LIN {X 0,Y 473.859,Z 535.178,A -85,B 0,C 180,E1 -7292.55,E2 -7292.55} C_VEL
LIN {X 0,Y 473.786,Z 533.185,A -85,B 0,C 180,E1 -7294.253,E2 -7294.253} C_VEL
LIN {X 0,Y 473.862,Z 529.069,A -85,B 0,C 180,E1 -7296.438,E2 -7296.438} C_VEL
LIN {X 0,Y 473.899,Z 524.706,A -85,B 0,C 180,E1 -7298.099,E2 -7298.099} C_VEL
LIN {X 0,Y 473.982,Z 519.093,A -85,B 0,C 180,E1 -7299.817,E2 -7299.817} C_VEL
LIN {X 0,Y 474.226,Z 512.098,A -85,B 0,C 180,E1 -7301.54,E2 -7301.54} C_VEL
LIN {X 0,Y 474.535,Z 503.681,A -85,B 0,C 180,E1 -7303.271,E2 -7303.271} C_VEL
LIN {X 0,Y 475.075,Z 493.63,A -85,B 0,C 180,E1 -7305.003,E2 -7305.003} C_VEL
LIN {X 0,Y 475.646,Z 483.269,A -85,B 0,C 180,E1 -7306.524,E2 -7306.524} C_VEL
LIN {X 0,Y 476.368,Z 471.017,A -85,B 0,C 180,E1 -7308.048,E2 -7308.048} C_VEL
LIN {X 0,Y 477.233,Z 457.973,A -85,B 0,C 180,E1 -7309.422,E2 -7309.422} C_VEL
LIN {X 0,Y 478.152,Z 444.159,A -85,B 0,C 180,E1 -7310.655,E2 -7310.655} C_VEL
LIN {X 0,Y 479.041,Z 429.731,A -85,B 0,C 180,E1 -7311.742,E2 -7311.742} C_VEL
LIN {X 0,Y 479.978,Z 414.203,A -85,B 0,C 180,E1 -7312.711,E2 -7312.711} C_VEL
LIN {X 0,Y 480.906,Z 398.033,A -85,B 0,C 180,E1 -7313.524,E2 -7313.524} C_VEL
LIN {X 0,Y 481.693,Z 381.393,A -85,B 0,C 180,E1 -7314.169,E2 -7314.169} C_VEL
LIN {X 0,Y 482.3,Z 365.314,A -85,B 0,C 180,E1 -7314.623,E2 -7314.623} C_VEL
LIN {X 0,Y 482.825,Z 343.034,A -85,B 0,C 180,E1 -7315.038,E2 -7315.038} C_VEL
LIN {X 0,Y 485.86,Z 178.498,A -85,B 0,C 180,E1 -7317.853,E2 -7317.853} C_VEL
LIN {X 0,Y 482.039,Z 153.132,A -85,B 0,C 180,E1 -7318.567,E2 -7318.567} C_VEL
LIN {X 0,Y 483.529,Z 126.486,A -85,B 0,C 180,E1 -7321.047,E2 -7321.047} C_VEL
LIN {X 0,Y 482.934,Z 123.424,A -85,B 0,C 180,E1 -7321.381,E2 -7321.381} C_VEL
LIN {X 0,Y 476.541,Z 103.71,A -85,B 0,C 180,E1 -7323.756,E2 -7323.756} C_VEL
LIN {X 0,Y 474.657,Z 97.672,A -85,B 0,C 180,E1 -7324.527,E2 -7324.527} C_VEL
LIN {X 0,Y 474.585,Z 97.681,A -85,B 0,C 180,E1 -7327.383,E2 -7327.383} C_VEL
LIN {X 0,Y 474.623,Z 97.676,A -85,B 0,C 180,E1 -7329.647,E2 -7329.647} C_VEL
LIN {X 0,Y 474.648,Z 97.673,A -85,B 0,C 180,E1 -7332.93,E2 -7332.93} C_VEL
LIN {X 0,Y 474.605,Z 97.678,A -85,B 0,C 180,E1 -7335.895,E2 -7335.895} C_VEL
LIN {X 0,Y 474.623,Z 97.672,A -85,B 0,C 180,E1 -7339.04,E2 -7339.04} C_VEL
LIN {X 0,Y 474.606,Z 97.675,A -85,B 0,C 180,E1 -7341.704,E2 -7341.704} C_VEL
LIN {X 0,Y 474.626,Z 97.674,A -85,B 0,C 180,E1 -7344.726,E2 -7344.726} C_VEL
LIN {X 0,Y 474.632,Z 97.674,A -85,B 0,C 180,E1 -7347.788,E2 -7347.788} C_VEL
LIN {X 0,Y 474.62,Z 97.673,A -85,B 0,C 180,E1 -7350.884,E2 -7350.884} C_VEL
LIN {X 0,Y 474.656,Z 97.67,A -85,B 0,C 180,E1 -7353.628,E2 -7353.628} C_VEL
LIN {X 0,Y 474.631,Z 97.672,A -85,B 0,C 180,E1 -7356.641,E2 -7356.641} C_VEL
LIN {X 0,Y 474.65,Z 97.675,A -85,B 0,C 180,E1 -7360.09,E2 -7360.09} C_VEL
LIN {X 0,Y 474.646,Z 97.669,A -85,B 0,C 180,E1 -7362.774,E2 -7362.774} C_VEL
LIN {X 0,Y 474.644,Z 97.672,A -85,B 0,C 180,E1 -7365.421,E2 -7365.421} C_VEL
LIN {X 0,Y 474.734,Z 97.663,A -85,B 0,C 180,E1 -7368.038,E2 -7368.038} C_VEL
LIN {X 0,Y 474.723,Z 97.663,A -85,B 0,C 180,E1 -7371.487,E2 -7371.487} C_VEL
LIN {X 0,Y 474.774,Z 97.657,A -85,B 0,C 180,E1 -7374.052,E2 -7374.052} C_VEL
LIN {X 0,Y 474.89,Z 97.644,A -85,B 0,C 180,E1 -7377.455,E2 -7377.455} C_VEL
LIN {X 0,Y 474.908,Z 97.64,A -85,B 0,C 180,E1 -7380,E2 -7380} C_VEL
LIN {X 0,Y 474.89,Z 97.638,A -85,B 0,C 180,E1 -7382.545,E2 -7382.545} C_VEL
LIN {X 0,Y 474.774,Z 97.656,A -85,B 0,C 180,E1 -7385.948,E2 -7385.948} C_VEL
LIN {X 0,Y 474.723,Z 97.659,A -85,B 0,C 180,E1 -7388.514,E2 -7388.514} C_VEL
LIN {X 0,Y 474.7,Z 97.664,A -85,B 0,C 180,E1 -7391.963,E2 -7391.963} C_VEL
LIN {X 0,Y 474.696,Z 97.67,A -85,B 0,C 180,E1 -7395.456,E2 -7395.456} C_VEL
LIN {X 0,Y 474.661,Z 97.671,A -85,B 0,C 180,E1 -7399.01,E2 -7399.01} C_VEL
LIN {X 0,Y 474.587,Z 97.679,A -85,B 0,C 180,E1 -7401.729,E2 -7401.729} C_VEL
LIN {X 0,Y 474.655,Z 97.668,A -85,B 0,C 180,E1 -7404.493,E2 -7404.493} C_VEL
LIN {X 0,Y 474.677,Z 97.671,A -85,B 0,C 180,E1 -7407.335,E2 -7407.335} C_VEL
LIN {X 0,Y 474.602,Z 97.674,A -85,B 0,C 180,E1 -7410.23,E2 -7410.23} C_VEL
LIN {X 0,Y 474.639,Z 97.676,A -85,B 0,C 180,E1 -7413.22,E2 -7413.22} C_VEL
LIN {X 0,Y 474.59,Z 97.677,A -85,B 0,C 180,E1 -7416.323,E2 -7416.323} C_VEL
LIN {X 0,Y 474.624,Z 97.672,A -85,B 0,C 180,E1 -7419.648,E2 -7419.648} C_VEL
LIN {X 0,Y 474.637,Z 97.678,A -85,B 0,C 180,E1 -7422.932,E2 -7422.932} C_VEL
LIN {X 0,Y 474.612,Z 97.673,A -85,B 0,C 180,E1 -7425.896,E2 -7425.896} C_VEL
LIN {X 0,Y 474.629,Z 97.676,A -85,B 0,C 180,E1 -7429.041,E2 -7429.041} C_VEL
LIN {X 0,Y 474.607,Z 97.674,A -85,B 0,C 180,E1 -7431.705,E2 -7431.705} C_VEL
LIN {X 0,Y 474.622,Z 97.68,A -85,B 0,C 180,E1 -7434.726,E2 -7434.726} C_VEL
LIN {X 0,Y 474.634,Z 97.671,A -85,B 0,C 180,E1 -7437.788,E2 -7437.788} C_VEL
LIN {X 0,Y 474.622,Z 97.676,A -85,B 0,C 180,E1 -7440.885,E2 -7440.885} C_VEL
LIN {X 0,Y 474.659,Z 97.667,A -85,B 0,C 180,E1 -7443.629,E2 -7443.629} C_VEL
LIN {X 0,Y 474.634,Z 97.676,A -85,B 0,C 180,E1 -7446.642,E2 -7446.642} C_VEL
LIN {X 0,Y 474.654,Z 97.672,A -85,B 0,C 180,E1 -7450.09,E2 -7450.09} C_VEL
LIN {X 0,Y 474.655,Z 97.668,A -85,B 0,C 180,E1 -7451.674,E2 -7451.674} C_VEL
LIN {X 0,Y 473.992,Z 97.759,A -85,B 0,C 180,E1 -7452.383,E2 -7452.383} C_VEL
LIN {X 0,Y 471.141,Z 98.108,A -85,B 0,C 180,E1 -7453.534,E2 -7453.534} C_VEL
LIN {X 0,Y 468.725,Z 98.413,A -85,B 0,C 180,E1 -7454.463,E2 -7454.463} C_VEL
LIN {X 0,Y 467.683,Z 98.537,A -85,B 0,C 180,E1 -7455.18,E2 -7455.18} C_VEL
LIN {X 0,Y 467.596,Z 98.547,A -85,B 0,C 180,E1 -7455.423,E2 -7455.423} C_VEL
LIN {X 0,Y 467.653,Z 98.542,A -85,B 0,C 180,E1 -7458.734,E2 -7458.734} C_VEL
LIN {X 0,Y 467.749,Z 98.536,A -85,B 0,C 180,E1 -7462.229,E2 -7462.229} C_VEL
LIN {X 0,Y 467.724,Z 98.532,A -85,B 0,C 180,E1 -7464.828,E2 -7464.828} C_VEL
LIN {X 0,Y 467.86,Z 98.515,A -85,B 0,C 180,E1 -7467.418,E2 -7467.418} C_VEL
LIN {X 0,Y 467.883,Z 98.519,A -85,B 0,C 180,E1 -7470.001,E2 -7470.001} C_VEL
LIN {X 0,Y 467.86,Z 98.516,A -85,B 0,C 180,E1 -7472.583,E2 -7472.583} C_VEL
LIN {X 0,Y 467.744,Z 98.536,A -85,B 0,C 180,E1 -7476.038,E2 -7476.038} C_VEL
LIN {X 0,Y 467.683,Z 98.537,A -85,B 0,C 180,E1 -7478.643,E2 -7478.643} C_VEL
LIN {X 0,Y 467.658,Z 98.544,A -85,B 0,C 180,E1 -7482.146,E2 -7482.146} C_VEL
LIN {X 0,Y 467.641,Z 98.549,A -85,B 0,C 180,E1 -7485.695,E2 -7485.695} C_VEL
LIN {X 0,Y 467.619,Z 98.544,A -85,B 0,C 180,E1 -7488.765,E2 -7488.765} C_VEL
LIN {X 0,Y 467.583,Z 98.552,A -85,B 0,C 180,E1 -7491.269,E2 -7491.269} C_VEL
LIN {X 0,Y 467.565,Z 98.555,A -85,B 0,C 180,E1 -7493.944,E2 -7493.944} C_VEL
LIN {X 0,Y 467.615,Z 98.545,A -85,B 0,C 180,E1 -7496.801,E2 -7496.801} C_VEL
LIN {X 0,Y 467.556,Z 98.557,A -85,B 0,C 180,E1 -7499.739,E2 -7499.739} C_VEL
LIN {X 0,Y 467.586,Z 98.549,A -85,B 0,C 180,E1 -7502.759,E2 -7502.759} C_VEL
LIN {X 0,Y 467.556,Z 98.555,A -85,B 0,C 180,E1 -7505.89,E2 -7505.89} C_VEL
LIN {X 0,Y 467.584,Z 98.554,A -85,B 0,C 180,E1 -7509.145,E2 -7509.145} C_VEL
LIN {X 0,Y 467.589,Z 98.548,A -85,B 0,C 180,E1 -7512.567,E2 -7512.567} C_VEL
LIN {X 0,Y 467.573,Z 98.555,A -85,B 0,C 180,E1 -7515.053,E2 -7515.053} C_VEL
LIN {X 0,Y 467.592,Z 98.553,A -85,B 0,C 180,E1 -7517.44,E2 -7517.44} C_VEL
LIN {X 0,Y 467.579,Z 98.553,A -85,B 0,C 180,E1 -7520.855,E2 -7520.855} C_VEL
LIN {X 0,Y 467.564,Z 98.554,A -85,B 0,C 180,E1 -7524.261,E2 -7524.261} C_VEL
LIN {X 0,Y 467.585,Z 98.554,A -85,B 0,C 180,E1 -7527.321,E2 -7527.321} C_VEL
LIN {X 0,Y 467.601,Z 98.553,A -85,B 0,C 180,E1 -7530.759,E2 -7530.759} C_VEL
LIN {X 0,Y 467.602,Z 98.611,A -85,B 0,C 180,E1 -7530.924,E2 -7530.924} C_VEL
LIN {X 0,Y 468.702,Z 101.51,A -85,B 0,C 180,E1 -7531.051,E2 -7531.051} C_VEL
LIN {X 0,Y 479.424,Z 123.039,A -85,B 0,C 180,E1 -7532.127,E2 -7532.127} C_VEL
LIN {X 0,Y 476.666,Z 259.884,A -85,B 0,C 180,E1 -7534.524,E2 -7534.524} C_VEL
LIN {X 0,Y 476.047,Z 294.28,A -85,B 0,C 180,E1 -7535.147,E2 -7535.147} C_VEL
LIN {X 0,Y 475.582,Z 310.876,A -85,B 0,C 180,E1 -7535.616,E2 -7535.616} C_VEL
LIN {X 0,Y 474.885,Z 327.698,A -85,B 0,C 180,E1 -7536.274,E2 -7536.274} C_VEL
LIN {X 0,Y 474.244,Z 341.789,A -85,B 0,C 180,E1 -7536.982,E2 -7536.982} C_VEL
LIN {X 0,Y 473.363,Z 356.419,A -85,B 0,C 180,E1 -7537.868,E2 -7537.868} C_VEL
LIN {X 0,Y 472.41,Z 371.384,A -85,B 0,C 180,E1 -7538.967,E2 -7538.967} C_VEL
LIN {X 0,Y 471.469,Z 385.104,A -85,B 0,C 180,E1 -7540.176,E2 -7540.176} C_VEL
LIN {X 0,Y 470.583,Z 397.739,A -85,B 0,C 180,E1 -7541.497,E2 -7541.497} C_VEL
LIN {X 0,Y 469.829,Z 408.765,A -85,B 0,C 180,E1 -7542.839,E2 -7542.839} C_VEL
LIN {X 0,Y 469.086,Z 419.478,A -85,B 0,C 180,E1 -7544.355,E2 -7544.355} C_VEL
LIN {X 0,Y 468.388,Z 429.934,A -85,B 0,C 180,E1 -7546.109,E2 -7546.109} C_VEL
LIN {X 0,Y 467.862,Z 438.612,A -85,B 0,C 180,E1 -7547.86,E2 -7547.86} C_VEL
LIN {X 0,Y 467.42,Z 445.822,A -85,B 0,C 180,E1 -7549.605,E2 -7549.605} C_VEL
LIN {X 0,Y 467.202,Z 451.766,A -85,B 0,C 180,E1 -7551.348,E2 -7551.348} C_VEL
LIN {X 0,Y 467.04,Z 457.016,A -85,B 0,C 180,E1 -7553.3,E2 -7553.3} C_VEL
LIN {X 0,Y 466.804,Z 460.099,A -85,B 0,C 180,E1 -7554.817,E2 -7554.817} C_VEL
LIN {X 0,Y 466.88,Z 462.699,A -85,B 0,C 180,E1 -7556.548,E2 -7556.548} C_VEL
LIN {X 0,Y 466.703,Z 464.258,A -85,B 0,C 180,E1 -7558.274,E2 -7558.274} C_VEL
LIN {X 0,Y 466.64,Z 464.913,A -85,B 0,C 180,E1 -7560,E2 -7560} C_VEL
LIN {X 0,Y 466.704,Z 464.491,A -85,B 0,C 180,E1 -7561.726,E2 -7561.726} C_VEL
LIN {X 0,Y 466.959,Z 463.165,A -85,B 0,C 180,E1 -7563.451,E2 -7563.451} C_VEL
LIN {X 0,Y 466.86,Z 460.78,A -85,B 0,C 180,E1 -7565.182,E2 -7565.182} C_VEL
LIN {X 0,Y 467.084,Z 457.398,A -85,B 0,C 180,E1 -7566.913,E2 -7566.913} C_VEL
LIN {X 0,Y 467.281,Z 452.9,A -85,B 0,C 180,E1 -7568.65,E2 -7568.65} C_VEL
LIN {X 0,Y 467.576,Z 447.202,A -85,B 0,C 180,E1 -7570.391,E2 -7570.391} C_VEL
LIN {X 0,Y 468.001,Z 440.246,A -85,B 0,C 180,E1 -7572.136,E2 -7572.136} C_VEL
LIN {X 0,Y 468.561,Z 431.809,A -85,B 0,C 180,E1 -7573.886,E2 -7573.886} C_VEL
LIN {X 0,Y 469.295,Z 421.61,A -85,B 0,C 180,E1 -7575.638,E2 -7575.638} C_VEL
LIN {X 0,Y 470.033,Z 411.025,A -85,B 0,C 180,E1 -7577.17,E2 -7577.17} C_VEL
LIN {X 0,Y 470.94,Z 398.417,A -85,B 0,C 180,E1 -7578.714,E2 -7578.714} C_VEL
LIN {X 0,Y 471.819,Z 385.64,A -85,B 0,C 180,E1 -7580.035,E2 -7580.035} C_VEL
LIN {X 0,Y 472.788,Z 371.749,A -85,B 0,C 180,E1 -7581.243,E2 -7581.243} C_VEL
LIN {X 0,Y 473.62,Z 358.252,A -85,B 0,C 180,E1 -7582.234,E2 -7582.234} C_VEL
LIN {X 0,Y 474.452,Z 343.088,A -85,B 0,C 180,E1 -7583.148,E2 -7583.148} C_VEL
LIN {X 0,Y 475.124,Z 327.956,A -85,B 0,C 180,E1 -7583.886,E2 -7583.886} C_VEL
LIN {X 0,Y 475.739,Z 311.166,A -85,B 0,C 180,E1 -7584.521,E2 -7584.521} C_VEL
LIN {X 0,Y 476.128,Z 296.356,A -85,B 0,C 180,E1 -7584.936,E2 -7584.936} C_VEL
LIN {X 0,Y 478.711,Z 200.411,A -85,B 0,C 180,E1 -7586.807,E2 -7586.807} C_VEL
LIN {X 0,Y 481.638,Z 124.343,A -85,B 0,C 180,E1 -7588.413,E2 -7588.413} C_VEL
LIN {X 0,Y 475.778,Z 113.062,A -85,B 0,C 180,E1 -7589.251,E2 -7589.251} C_VEL
LIN {X 0,Y 471.346,Z 105.664,A -85,B 0,C 180,E1 -7589.905,E2 -7589.905} C_VEL
LIN {X 0,Y 469.754,Z 102.867,A -85,B 0,C 180,E1 -7590.156,E2 -7590.156} C_VEL
LIN {X 0,Y 468.059,Z 100.482,A -85,B 0,C 180,E1 -7590.418,E2 -7590.418} C_VEL
LIN {X 0,Y 467.546,Z 98.562,A -85,B 0,C 180,E1 -7590.552,E2 -7590.552} C_VEL
LIN {X 0,Y 467.571,Z 98.556,A -85,B 0,C 180,E1 -7593.789,E2 -7593.789} C_VEL
LIN {X 0,Y 467.525,Z 98.563,A -85,B 0,C 180,E1 -7596.962,E2 -7596.962} C_VEL
LIN {X 0,Y 467.577,Z 98.555,A -85,B 0,C 180,E1 -7599.953,E2 -7599.953} C_VEL
LIN {X 0,Y 467.588,Z 98.555,A -85,B 0,C 180,E1 -7602.567,E2 -7602.567} C_VEL
LIN {X 0,Y 467.568,Z 98.555,A -85,B 0,C 180,E1 -7605.052,E2 -7605.052} C_VEL
LIN {X 0,Y 467.591,Z 98.554,A -85,B 0,C 180,E1 -7607.439,E2 -7607.439} C_VEL
LIN {X 0,Y 467.583,Z 98.555,A -85,B 0,C 180,E1 -7610.855,E2 -7610.855} C_VEL
LIN {X 0,Y 467.561,Z 98.702,A -85,B 0,C 180,E1 -7613.844,E2 -7613.844} C_VEL
LIN {X 0,Y 470.978,Z 107.315,A -85,B 0,C 180,E1 -7615.455,E2 -7615.455} C_VEL
LIN {X 0,Y 474.497,Z 117.269,A -85,B 0,C 180,E1 -7617.075,E2 -7617.075} C_VEL
LIN {X 0,Y 477.215,Z 126.936,A -85,B 0,C 180,E1 -7618.452,E2 -7618.452} C_VEL
LIN {X 0,Y 477.057,Z 131.636,A -85,B 0,C 180,E1 -7618.961,E2 -7618.961} C_VEL
LIN {X 0,Y 475.985,Z 144.526,A -85,B 0,C 180,E1 -7620.279,E2 -7620.279} C_VEL
LIN {X 0,Y 479.377,Z 168.319,A -85,B 0,C 180,E1 -7621.187,E2 -7621.187} C_VEL
LIN {X 0,Y 480.601,Z 180.632,A -85,B 0,C 180,E1 -7621.582,E2 -7621.582} C_VEL
LIN {X 0,Y 477.522,Z 271.244,A -85,B 0,C 180,E1 -7623.416,E2 -7623.416} C_VEL
LIN {X 0,Y 475.395,Z 359.016,A -85,B 0,C 180,E1 -7625.081,E2 -7625.081} C_VEL
LIN {X 0,Y 474.661,Z 376.224,A -85,B 0,C 180,E1 -7625.565,E2 -7625.565} C_VEL
LIN {X 0,Y 473.732,Z 394.362,A -85,B 0,C 180,E1 -7626.271,E2 -7626.271} C_VEL
LIN {X 0,Y 472.797,Z 410.384,A -85,B 0,C 180,E1 -7627.077,E2 -7627.077} C_VEL
LIN {X 0,Y 471.845,Z 425.719,A -85,B 0,C 180,E1 -7628.024,E2 -7628.024} C_VEL
LIN {X 0,Y 470.925,Z 440.572,A -85,B 0,C 180,E1 -7629.126,E2 -7629.126} C_VEL
LIN {X 0,Y 469.973,Z 455.118,A -85,B 0,C 180,E1 -7630.407,E2 -7630.407} C_VEL
LIN {X 0,Y 469.24,Z 467.347,A -85,B 0,C 180,E1 -7631.667,E2 -7631.667} C_VEL
LIN {X 0,Y 468.512,Z 480.115,A -85,B 0,C 180,E1 -7633.216,E2 -7633.216} C_VEL
LIN {X 0,Y 467.957,Z 490.942,A -85,B 0,C 180,E1 -7634.762,E2 -7634.762} C_VEL
LIN {X 0,Y 467.439,Z 501.436,A -85,B 0,C 180,E1 -7636.523,E2 -7636.523} C_VEL
LIN {X 0,Y 467.153,Z 510.275,A -85,B 0,C 180,E1 -7638.294,E2 -7638.294} C_VEL
LIN {X 0,Y 466.896,Z 517.51,A -85,B 0,C 180,E1 -7640.031,E2 -7640.031} C_VEL
LIN {X 0,Y 466.813,Z 524.699,A -85,B 0,C 180,E1 -7642.212,E2 -7642.212} C_VEL
LIN {X 0,Y 466.803,Z 529.037,A -85,B 0,C 180,E1 -7643.95,E2 -7643.95} C_VEL
LIN {X 0,Y 466.715,Z 532.292,A -85,B 0,C 180,E1 -7645.681,E2 -7645.681} C_VEL
LIN {X 0,Y 466.805,Z 534.444,A -85,B 0,C 180,E1 -7647.411,E2 -7647.411} C_VEL
LIN {X 0,Y 466.632,Z 535.538,A -85,B 0,C 180,E1 -7649.136,E2 -7649.136} C_VEL
LIN {X 0,Y 466.63,Z 535.61,A -85,B 0,C 180,E1 -7650.862,E2 -7650.862} C_VEL
LIN {X 0,Y 466.799,Z 534.646,A -85,B 0,C 180,E1 -7652.588,E2 -7652.588} C_VEL
LIN {X 0,Y 466.694,Z 532.647,A -85,B 0,C 180,E1 -7654.318,E2 -7654.318} C_VEL
LIN {X 0,Y 466.786,Z 528.732,A -85,B 0,C 180,E1 -7656.434,E2 -7656.434} C_VEL
LIN {X 0,Y 466.83,Z 524.128,A -85,B 0,C 180,E1 -7658.222,E2 -7658.222} C_VEL
LIN {X 0,Y 466.893,Z 518.484,A -85,B 0,C 180,E1 -7659.968,E2 -7659.968} C_VEL
LIN {X 0,Y 467.185,Z 511.463,A -85,B 0,C 180,E1 -7661.717,E2 -7661.717} C_VEL
LIN {X 0,Y 467.489,Z 503,A -85,B 0,C 180,E1 -7663.474,E2 -7663.474} C_VEL
LIN {X 0,Y 468.062,Z 492.885,A -85,B 0,C 180,E1 -7665.234,E2 -7665.234} C_VEL
LIN {X 0,Y 468.685,Z 482.45,A -85,B 0,C 180,E1 -7666.777,E2 -7666.777} C_VEL
LIN {X 0,Y 469.446,Z 470.13,A -85,B 0,C 180,E1 -7668.323,E2 -7668.323} C_VEL
LIN {X 0,Y 470.42,Z 456.7,A -85,B 0,C 180,E1 -7669.745,E2 -7669.745} C_VEL
LIN {X 0,Y 471.338,Z 443.065,A -85,B 0,C 180,E1 -7670.968,E2 -7670.968} C_VEL
LIN {X 0,Y 472.315,Z 428.512,A -85,B 0,C 180,E1 -7672.068,E2 -7672.068} C_VEL
LIN {X 0,Y 473.281,Z 413.462,A -85,B 0,C 180,E1 -7673.014,E2 -7673.014} C_VEL
LIN {X 0,Y 474.227,Z 397.654,A -85,B 0,C 180,E1 -7673.818,E2 -7673.818} C_VEL
LIN {X 0,Y 475.086,Z 380.298,A -85,B 0,C 180,E1 -7674.498,E2 -7674.498} C_VEL
LIN {X 0,Y 475.751,Z 362.876,A -85,B 0,C 180,E1 -7674.985,E2 -7674.985} C_VEL
LIN {X 0,Y 476.47,Z 329.67,A -85,B 0,C 180,E1 -7675.579,E2 -7675.579} C_VEL
LIN {X 0,Y 479.49,Z 179.426,A -85,B 0,C 180,E1 -7678.208,E2 -7678.208} C_VEL
LIN {X 0,Y 475.516,Z 152.621,A -85,B 0,C 180,E1 -7678.985,E2 -7678.985} C_VEL
LIN {X 0,Y 476.95,Z 128.263,A -85,B 0,C 180,E1 -7681.28,E2 -7681.28} C_VEL
LIN {X 0,Y 473.296,Z 116.03,A -85,B 0,C 180,E1 -7682.734,E2 -7682.734} C_VEL
LIN {X 0,Y 467.603,Z 98.552,A -85,B 0,C 180,E1 -7684.927,E2 -7684.927} C_VEL
LIN {X 0,Y 467.557,Z 98.56,A -85,B 0,C 180,E1 -7688.59,E2 -7688.59} C_VEL
LIN {X 0,Y 467.579,Z 98.552,A -85,B 0,C 180,E1 -7691.402,E2 -7691.402} C_VEL
LIN {X 0,Y 467.57,Z 98.553,A -85,B 0,C 180,E1 -7693.823,E2 -7693.823} C_VEL
LIN {X 0,Y 467.551,Z 98.56,A -85,B 0,C 180,E1 -7696.255,E2 -7696.255} C_VEL
LIN {X 0,Y 467.573,Z 98.553,A -85,B 0,C 180,E1 -7698.723,E2 -7698.723} C_VEL
LIN {X 0,Y 467.562,Z 98.555,A -85,B 0,C 180,E1 -7701.955,E2 -7701.955} C_VEL
LIN {X 0,Y 467.564,Z 98.551,A -85,B 0,C 180,E1 -7705.168,E2 -7705.168} C_VEL
LIN {X 0,Y 467.579,Z 98.556,A -85,B 0,C 180,E1 -7708.26,E2 -7708.26} C_VEL
LIN {X 0,Y 467.573,Z 98.55,A -85,B 0,C 180,E1 -7711.25,E2 -7711.25} C_VEL
LIN {X 0,Y 467.611,Z 98.545,A -85,B 0,C 180,E1 -7713.2,E2 -7713.2} C_VEL
LIN {X 0,Y 467.588,Z 98.551,A -85,B 0,C 180,E1 -7716.468,E2 -7716.468} C_VEL
LIN {X 0,Y 467.618,Z 98.55,A -85,B 0,C 180,E1 -7719.777,E2 -7719.777} C_VEL
LIN {X 0,Y 467.604,Z 98.548,A -85,B 0,C 180,E1 -7722.507,E2 -7722.507} C_VEL
LIN {X 0,Y 467.602,Z 98.547,A -85,B 0,C 180,E1 -7725.196,E2 -7725.196} C_VEL
LIN {X 0,Y 467.678,Z 98.545,A -85,B 0,C 180,E1 -7727.855,E2 -7727.855} C_VEL
LIN {X 0,Y 467.677,Z 98.54,A -85,B 0,C 180,E1 -7731.357,E2 -7731.357} C_VEL
LIN {X 0,Y 467.739,Z 98.534,A -85,B 0,C 180,E1 -7733.963,E2 -7733.963} C_VEL
LIN {X 0,Y 467.855,Z 98.519,A -85,B 0,C 180,E1 -7737.417,E2 -7737.417} C_VEL
LIN {X 0,Y 467.878,Z 98.515,A -85,B 0,C 180,E1 -7740,E2 -7740} C_VEL
LIN {X 0,Y 467.856,Z 98.515,A -85,B 0,C 180,E1 -7742.583,E2 -7742.583} C_VEL
LIN {X 0,Y 467.739,Z 98.531,A -85,B 0,C 180,E1 -7746.038,E2 -7746.038} C_VEL
LIN {X 0,Y 467.677,Z 98.537,A -85,B 0,C 180,E1 -7748.643,E2 -7748.643} C_VEL
LIN {X 0,Y 467.651,Z 98.541,A -85,B 0,C 180,E1 -7752.146,E2 -7752.146} C_VEL
LIN {X 0,Y 467.635,Z 98.546,A -85,B 0,C 180,E1 -7755.695,E2 -7755.695} C_VEL
LIN {X 0,Y 467.614,Z 98.547,A -85,B 0,C 180,E1 -7758.765,E2 -7758.765} C_VEL
LIN {X 0,Y 467.577,Z 98.558,A -85,B 0,C 180,E1 -7761.269,E2 -7761.269} C_VEL
LIN {X 0,Y 467.569,Z 98.551,A -85,B 0,C 180,E1 -7763.943,E2 -7763.943} C_VEL
LIN {X 0,Y 467.612,Z 98.548,A -85,B 0,C 180,E1 -7766.801,E2 -7766.801} C_VEL
LIN {X 0,Y 467.55,Z 98.554,A -85,B 0,C 180,E1 -7769.738,E2 -7769.738} C_VEL
LIN {X 0,Y 467.58,Z 98.553,A -85,B 0,C 180,E1 -7772.759,E2 -7772.759} C_VEL
LIN {X 0,Y 467.553,Z 98.553,A -85,B 0,C 180,E1 -7775.89,E2 -7775.89} C_VEL
LIN {X 0,Y 467.579,Z 98.555,A -85,B 0,C 180,E1 -7779.145,E2 -7779.145} C_VEL
LIN {X 0,Y 467.583,Z 98.553,A -85,B 0,C 180,E1 -7782.567,E2 -7782.567} C_VEL
LIN {X 0,Y 467.568,Z 98.556,A -85,B 0,C 180,E1 -7785.054,E2 -7785.054} C_VEL
LIN {X 0,Y 467.585,Z 98.549,A -85,B 0,C 180,E1 -7787.44,E2 -7787.44} C_VEL
LIN {X 0,Y 467.589,Z 98.555,A -85,B 0,C 180,E1 -7790.857,E2 -7790.857} C_VEL
LIN {X 0,Y 467.557,Z 98.555,A -85,B 0,C 180,E1 -7794.261,E2 -7794.261} C_VEL
LIN {X 0,Y 467.579,Z 98.55,A -85,B 0,C 180,E1 -7797.321,E2 -7797.321} C_VEL
LIN {X 0,Y 467.568,Z 98.557,A -85,B 0,C 180,E1 -7800.668,E2 -7800.668} C_VEL
LIN {X 0,Y 467.614,Z 98.546,A -85,B 0,C 180,E1 -7803.2,E2 -7803.2} C_VEL
LIN {X 0,Y 467.591,Z 98.556,A -85,B 0,C 180,E1 -7806.469,E2 -7806.469} C_VEL
LIN {X 0,Y 467.622,Z 98.545,A -85,B 0,C 180,E1 -7809.778,E2 -7809.778} C_VEL
LIN {X 0,Y 467.608,Z 98.552,A -85,B 0,C 180,E1 -7812.507,E2 -7812.507} C_VEL
LIN {X 0,Y 467.596,Z 98.547,A -85,B 0,C 180,E1 -7815.423,E2 -7815.423} C_VEL
LIN {X 0,Y 466.926,Z 98.637,A -85,B 0,C 180,E1 -7816.142,E2 -7816.142} C_VEL
LIN {X 0,Y 464.083,Z 98.987,A -85,B 0,C 180,E1 -7817.31,E2 -7817.31} C_VEL
LIN {X 0,Y 461.684,Z 99.292,A -85,B 0,C 180,E1 -7818.253,E2 -7818.253} C_VEL
LIN {X 0,Y 460.658,Z 99.413,A -85,B 0,C 180,E1 -7818.98,E2 -7818.98} C_VEL
LIN {X 0,Y 460.576,Z 99.422,A -85,B 0,C 180,E1 -7819.227,E2 -7819.227} C_VEL
LIN {X 0,Y 460.72,Z 99.407,A -85,B 0,C 180,E1 -7822.539,E2 -7822.539} C_VEL
LIN {X 0,Y 460.697,Z 99.408,A -85,B 0,C 180,E1 -7824.749,E2 -7824.749} C_VEL
LIN {X 0,Y 460.801,Z 99.394,A -85,B 0,C 180,E1 -7827.378,E2 -7827.378} C_VEL
LIN {X 0,Y 460.853,Z 99.394,A -85,B 0,C 180,E1 -7830.001,E2 -7830.001} C_VEL
LIN {X 0,Y 460.801,Z 99.395,A -85,B 0,C 180,E1 -7832.623,E2 -7832.623} C_VEL
LIN {X 0,Y 460.71,Z 99.411,A -85,B 0,C 180,E1 -7836.13,E2 -7836.13} C_VEL
LIN {X 0,Y 460.63,Z 99.415,A -85,B 0,C 180,E1 -7838.777,E2 -7838.777} C_VEL
LIN {X 0,Y 460.615,Z 99.418,A -85,B 0,C 180,E1 -7842.445,E2 -7842.445} C_VEL
LIN {X 0,Y 460.602,Z 99.423,A -85,B 0,C 180,E1 -7845.998,E2 -7845.998} C_VEL
LIN {X 0,Y 460.573,Z 99.422,A -85,B 0,C 180,E1 -7848.902,E2 -7848.902} C_VEL
LIN {X 0,Y 460.518,Z 99.434,A -85,B 0,C 180,E1 -7851.486,E2 -7851.486} C_VEL
LIN {X 0,Y 460.533,Z 99.428,A -85,B 0,C 180,E1 -7854.333,E2 -7854.333} C_VEL
LIN {X 0,Y 460.591,Z 99.425,A -85,B 0,C 180,E1 -7857.748,E2 -7857.748} C_VEL
LIN {X 0,Y 460.524,Z 99.433,A -85,B 0,C 180,E1 -7861.283,E2 -7861.283} C_VEL
LIN {X 0,Y 460.534,Z 99.427,A -85,B 0,C 180,E1 -7864.506,E2 -7864.506} C_VEL
LIN {X 0,Y 460.503,Z 99.436,A -85,B 0,C 180,E1 -7867.624,E2 -7867.624} C_VEL
LIN {X 0,Y 460.544,Z 99.426,A -85,B 0,C 180,E1 -7870.27,E2 -7870.27} C_VEL
LIN {X 0,Y 460.511,Z 99.437,A -85,B 0,C 180,E1 -7873.375,E2 -7873.375} C_VEL
LIN {X 0,Y 460.503,Z 99.432,A -85,B 0,C 180,E1 -7876.625,E2 -7876.625} C_VEL
LIN {X 0,Y 460.542,Z 99.428,A -85,B 0,C 180,E1 -7879.731,E2 -7879.731} C_VEL
LIN {X 0,Y 460.503,Z 99.432,A -85,B 0,C 180,E1 -7882.524,E2 -7882.524} C_VEL
LIN {X 0,Y 460.551,Z 99.428,A -85,B 0,C 180,E1 -7885.624,E2 -7885.624} C_VEL
LIN {X 0,Y 460.541,Z 99.432,A -85,B 0,C 180,E1 -7888.745,E2 -7888.745} C_VEL
LIN {X 0,Y 460.527,Z 99.434,A -85,B 0,C 180,E1 -7890.475,E2 -7890.475} C_VEL
LIN {X 0,Y 461.699,Z 102.547,A -85,B 0,C 180,E1 -7890.627,E2 -7890.627} C_VEL
LIN {X 0,Y 473.041,Z 125.211,A -85,B 0,C 180,E1 -7891.788,E2 -7891.788} C_VEL
LIN {X 0,Y 469.882,Z 274.054,A -85,B 0,C 180,E1 -7894.443,E2 -7894.443} C_VEL
LIN {X 0,Y 469.42,Z 295.634,A -85,B 0,C 180,E1 -7894.861,E2 -7894.861} C_VEL
LIN {X 0,Y 468.936,Z 311.955,A -85,B 0,C 180,E1 -7895.336,E2 -7895.336} C_VEL
LIN {X 0,Y 468.252,Z 327.992,A -85,B 0,C 180,E1 -7895.976,E2 -7895.976} C_VEL
LIN {X 0,Y 467.562,Z 342.083,A -85,B 0,C 180,E1 -7896.691,E2 -7896.691} C_VEL
LIN {X 0,Y 466.595,Z 357.58,A -85,B 0,C 180,E1 -7897.646,E2 -7897.646} C_VEL
LIN {X 0,Y 465.593,Z 372.421,A -85,B 0,C 180,E1 -7898.76,E2 -7898.76} C_VEL
LIN {X 0,Y 464.648,Z 385.675,A -85,B 0,C 180,E1 -7899.947,E2 -7899.947} C_VEL
LIN {X 0,Y 463.781,Z 397.667,A -85,B 0,C 180,E1 -7901.215,E2 -7901.215} C_VEL
LIN {X 0,Y 462.856,Z 410.292,A -85,B 0,C 180,E1 -7902.778,E2 -7902.778} C_VEL
LIN {X 0,Y 462.074,Z 420.993,A -85,B 0,C 180,E1 -7904.337,E2 -7904.337} C_VEL
LIN {X 0,Y 461.443,Z 430.141,A -85,B 0,C 180,E1 -7905.896,E2 -7905.896} C_VEL
LIN {X 0,Y 460.869,Z 438.893,A -85,B 0,C 180,E1 -7907.673,E2 -7907.673} C_VEL
LIN {X 0,Y 460.402,Z 446.172,A -85,B 0,C 180,E1 -7909.445,E2 -7909.445} C_VEL
LIN {X 0,Y 460.181,Z 452.167,A -85,B 0,C 180,E1 -7911.215,E2 -7911.215} C_VEL
LIN {X 0,Y 459.995,Z 457.622,A -85,B 0,C 180,E1 -7913.268,E2 -7913.268} C_VEL
LIN {X 0,Y 459.744,Z 460.575,A -85,B 0,C 180,E1 -7914.737,E2 -7914.737} C_VEL
LIN {X 0,Y 459.808,Z 463.199,A -85,B 0,C 180,E1 -7916.495,E2 -7916.495} C_VEL
LIN {X 0,Y 459.643,Z 464.786,A -85,B 0,C 180,E1 -7918.248,E2 -7918.248} C_VEL
LIN {X 0,Y 459.569,Z 465.459,A -85,B 0,C 180,E1 -7920,E2 -7920} C_VEL
LIN {X 0,Y 459.644,Z 465.052,A -85,B 0,C 180,E1 -7921.752,E2 -7921.752} C_VEL
LIN {X 0,Y 459.894,Z 463.739,A -85,B 0,C 180,E1 -7923.504,E2 -7923.504} C_VEL
LIN {X 0,Y 459.801,Z 461.362,A -85,B 0,C 180,E1 -7925.262,E2 -7925.262} C_VEL
LIN {X 0,Y 460.049,Z 457.977,A -85,B 0,C 180,E1 -7927.02,E2 -7927.02} C_VEL
LIN {X 0,Y 460.274,Z 453.482,A -85,B 0,C 180,E1 -7928.783,E2 -7928.783} C_VEL
LIN {X 0,Y 460.599,Z 447.785,A -85,B 0,C 180,E1 -7930.55,E2 -7930.55} C_VEL
LIN {X 0,Y 461.05,Z 440.817,A -85,B 0,C 180,E1 -7932.322,E2 -7932.322} C_VEL
LIN {X 0,Y 461.671,Z 432.38,A -85,B 0,C 180,E1 -7934.097,E2 -7934.097} C_VEL
LIN {X 0,Y 462.452,Z 422.171,A -85,B 0,C 180,E1 -7935.876,E2 -7935.876} C_VEL
LIN {X 0,Y 463.215,Z 411.687,A -85,B 0,C 180,E1 -7937.416,E2 -7937.416} C_VEL
LIN {X 0,Y 464.206,Z 398.965,A -85,B 0,C 180,E1 -7938.996,E2 -7938.996} C_VEL
LIN {X 0,Y 465.162,Z 386.186,A -85,B 0,C 180,E1 -7940.334,E2 -7940.334} C_VEL
LIN {X 0,Y 466.183,Z 372.292,A -85,B 0,C 180,E1 -7941.559,E2 -7941.559} C_VEL
LIN {X 0,Y 467.06,Z 358.817,A -85,B 0,C 180,E1 -7942.563,E2 -7942.563} C_VEL
LIN {X 0,Y 468.035,Z 342.591,A -85,B 0,C 180,E1 -7943.551,E2 -7943.551} C_VEL
LIN {X 0,Y 468.792,Z 326.115,A -85,B 0,C 180,E1 -7944.347,E2 -7944.347} C_VEL
LIN {X 0,Y 469.398,Z 309.421,A -85,B 0,C 180,E1 -7944.963,E2 -7944.963} C_VEL
LIN {X 0,Y 469.801,Z 293.52,A -85,B 0,C 180,E1 -7945.384,E2 -7945.384} C_VEL
LIN {X 0,Y 472.415,Z 207.105,A -85,B 0,C 180,E1 -7947.117,E2 -7947.117} C_VEL
LIN {X 0,Y 475.858,Z 127.331,A -85,B 0,C 180,E1 -7948.853,E2 -7948.853} C_VEL
LIN {X 0,Y 474.92,Z 124.982,A -85,B 0,C 180,E1 -7949.005,E2 -7949.005} C_VEL
LIN {X 0,Y 469.47,Z 114.752,A -85,B 0,C 180,E1 -7949.831,E2 -7949.831} C_VEL
LIN {X 0,Y 465.18,Z 107.699,A -85,B 0,C 180,E1 -7950.513,E2 -7950.513} C_VEL
LIN {X 0,Y 462.81,Z 103.847,A -85,B 0,C 180,E1 -7950.91,E2 -7950.91} C_VEL
LIN {X 0,Y 461.013,Z 101.308,A -85,B 0,C 180,E1 -7951.212,E2 -7951.212} C_VEL
LIN {X 0,Y 460.635,Z 100.117,A -85,B 0,C 180,E1 -7951.305,E2 -7951.305} C_VEL
LIN {X 0,Y 460.529,Z 99.435,A -85,B 0,C 180,E1 -7951.511,E2 -7951.511} C_VEL
LIN {X 0,Y 460.524,Z 99.435,A -85,B 0,C 180,E1 -7954.503,E2 -7954.503} C_VEL
LIN {X 0,Y 460.5,Z 99.437,A -85,B 0,C 180,E1 -7957.623,E2 -7957.623} C_VEL
LIN {X 0,Y 460.54,Z 99.433,A -85,B 0,C 180,E1 -7960.268,E2 -7960.268} C_VEL
LIN {X 0,Y 460.5,Z 99.436,A -85,B 0,C 180,E1 -7963.375,E2 -7963.375} C_VEL
LIN {X 0,Y 460.5,Z 99.437,A -85,B 0,C 180,E1 -7966.624,E2 -7966.624} C_VEL
LIN {X 0,Y 460.543,Z 99.433,A -85,B 0,C 180,E1 -7969.73,E2 -7969.73} C_VEL
LIN {X 0,Y 460.513,Z 99.437,A -85,B 0,C 180,E1 -7972.927,E2 -7972.927} C_VEL
LIN {X 0,Y 461.616,Z 102.442,A -85,B 0,C 180,E1 -7973.575,E2 -7973.575} C_VEL
LIN {X 0,Y 464.786,Z 110.237,A -85,B 0,C 180,E1 -7975.115,E2 -7975.115} C_VEL
LIN {X 0,Y 468.28,Z 120.101,A -85,B 0,C 180,E1 -7976.793,E2 -7976.793} C_VEL
LIN {X 0,Y 471.011,Z 130.17,A -85,B 0,C 180,E1 -7978.266,E2 -7978.266} C_VEL
LIN {X 0,Y 469.895,Z 143.496,A -85,B 0,C 180,E1 -7979.678,E2 -7979.678} C_VEL
LIN {X 0,Y 472.756,Z 163.249,A -85,B 0,C 180,E1 -7980.488,E2 -7980.488} C_VEL
LIN {X 0,Y 474.638,Z 181.845,A -85,B 0,C 180,E1 -7981.135,E2 -7981.135} C_VEL
LIN {X 0,Y 471.286,Z 271.227,A -85,B 0,C 180,E1 -7983.006,E2 -7983.006} C_VEL
LIN {X 0,Y 468.952,Z 358.324,A -85,B 0,C 180,E1 -7984.715,E2 -7984.715} C_VEL
LIN {X 0,Y 468.104,Z 376.106,A -85,B 0,C 180,E1 -7985.229,E2 -7985.229} C_VEL
LIN {X 0,Y 467.167,Z 393.412,A -85,B 0,C 180,E1 -7985.916,E2 -7985.916} C_VEL
LIN {X 0,Y 466.077,Z 410.659,A -85,B 0,C 180,E1 -7986.8,E2 -7986.8} C_VEL
LIN {X 0,Y 465.018,Z 426.379,A -85,B 0,C 180,E1 -7987.8,E2 -7987.8} C_VEL
LIN {X 0,Y 464.058,Z 440.985,A -85,B 0,C 180,E1 -7988.919,E2 -7988.919} C_VEL
LIN {X 0,Y 463.068,Z 455.314,A -85,B 0,C 180,E1 -7990.215,E2 -7990.215} C_VEL
LIN {X 0,Y 462.2,Z 468.381,A -85,B 0,C 180,E1 -7991.608,E2 -7991.608} C_VEL
LIN {X 0,Y 461.456,Z 480.943,A -85,B 0,C 180,E1 -7993.179,E2 -7993.179} C_VEL
LIN {X 0,Y 460.884,Z 491.605,A -85,B 0,C 180,E1 -7994.749,E2 -7994.749} C_VEL
LIN {X 0,Y 460.416,Z 500.691,A -85,B 0,C 180,E1 -7996.314,E2 -7996.314} C_VEL
LIN {X 0,Y 460.076,Z 509.866,A -85,B 0,C 180,E1 -7998.178,E2 -7998.178} C_VEL
LIN {X 0,Y 459.823,Z 516.845,A -85,B 0,C 180,E1 -7999.876,E2 -7999.876} C_VEL
LIN {X 0,Y 459.75,Z 524.077,A -85,B 0,C 180,E1 -8002.092,E2 -8002.092} C_VEL
LIN {X 0,Y 459.726,Z 528.442,A -85,B 0,C 180,E1 -8003.856,E2 -8003.856} C_VEL
LIN {X 0,Y 459.627,Z 531.72,A -85,B 0,C 180,E1 -8005.615,E2 -8005.615} C_VEL
LIN {X 0,Y 459.73,Z 533.891,A -85,B 0,C 180,E1 -8007.371,E2 -8007.371} C_VEL
LIN {X 0,Y 459.564,Z 534.997,A -85,B 0,C 180,E1 -8009.123,E2 -8009.123} C_VEL
LIN {X 0,Y 459.562,Z 535.076,A -85,B 0,C 180,E1 -8010.876,E2 -8010.876} C_VEL
LIN {X 0,Y 459.71,Z 534.108,A -85,B 0,C 180,E1 -8012.628,E2 -8012.628} C_VEL
LIN {X 0,Y 459.605,Z 532.105,A -85,B 0,C 180,E1 -8014.384,E2 -8014.384} C_VEL
LIN {X 0,Y 459.709,Z 528.39,A -85,B 0,C 180,E1 -8016.429,E2 -8016.429} C_VEL
LIN {X 0,Y 459.743,Z 523.535,A -85,B 0,C 180,E1 -8018.35,E2 -8018.35} C_VEL
LIN {X 0,Y 459.82,Z 517.855,A -85,B 0,C 180,E1 -8020.123,E2 -8020.123} C_VEL
LIN {X 0,Y 460.109,Z 511.075,A -85,B 0,C 180,E1 -8021.834,E2 -8021.834} C_VEL
LIN {X 0,Y 460.466,Z 502.276,A -85,B 0,C 180,E1 -8023.684,E2 -8023.684} C_VEL
LIN {X 0,Y 461.041,Z 492.093,A -85,B 0,C 180,E1 -8025.471,E2 -8025.471} C_VEL
LIN {X 0,Y 461.709,Z 481.588,A -85,B 0,C 180,E1 -8027.038,E2 -8027.038} C_VEL
LIN {X 0,Y 462.535,Z 469.211,A -85,B 0,C 180,E1 -8028.607,E2 -8028.607} C_VEL
LIN {X 0,Y 463.557,Z 455.588,A -85,B 0,C 180,E1 -8030.059,E2 -8030.059} C_VEL
LIN {X 0,Y 464.534,Z 441.902,A -85,B 0,C 180,E1 -8031.29,E2 -8031.29} C_VEL
LIN {X 0,Y 465.473,Z 428.787,A -85,B 0,C 180,E1 -8032.293,E2 -8032.293} C_VEL
LIN {X 0,Y 466.508,Z 413.553,A -85,B 0,C 180,E1 -8033.27,E2 -8033.27} C_VEL
LIN {X 0,Y 467.512,Z 397.084,A -85,B 0,C 180,E1 -8034.123,E2 -8034.123} C_VEL
LIN {X 0,Y 468.406,Z 379.746,A -85,B 0,C 180,E1 -8034.811,E2 -8034.811} C_VEL
LIN {X 0,Y 469.134,Z 362.376,A -85,B 0,C 180,E1 -8035.303,E2 -8035.303} C_VEL
LIN {X 0,Y 469.88,Z 329.685,A -85,B 0,C 180,E1 -8035.899,E2 -8035.899} C_VEL
LIN {X 0,Y 473.094,Z 180.14,A -85,B 0,C 180,E1 -8038.573,E2 -8038.573} C_VEL
LIN {X 0,Y 468.95,Z 152.396,A -85,B 0,C 180,E1 -8039.384,E2 -8039.384} C_VEL
LIN {X 0,Y 470.239,Z 129.495,A -85,B 0,C 180,E1 -8041.582,E2 -8041.582} C_VEL
LIN {X 0,Y 464.139,Z 110.541,A -85,B 0,C 180,E1 -8043.912,E2 -8043.912} C_VEL
LIN {X 0,Y 460.546,Z 99.431,A -85,B 0,C 180,E1 -8045.333,E2 -8045.333} C_VEL
LIN {X 0,Y 460.54,Z 99.432,A -85,B 0,C 180,E1 -8048.897,E2 -8048.897} C_VEL
LIN {X 0,Y 460.542,Z 99.433,A -85,B 0,C 180,E1 -8052.178,E2 -8052.178} C_VEL
LIN {X 0,Y 460.512,Z 99.432,A -85,B 0,C 180,E1 -8055.411,E2 -8055.411} C_VEL
LIN {X 0,Y 460.527,Z 99.435,A -85,B 0,C 180,E1 -8058.397,E2 -8058.397} C_VEL
LIN {X 0,Y 460.522,Z 99.428,A -85,B 0,C 180,E1 -8061.267,E2 -8061.267} C_VEL
LIN {X 0,Y 460.509,Z 99.434,A -85,B 0,C 180,E1 -8064.554,E2 -8064.554} C_VEL
LIN {X 0,Y 460.527,Z 99.43,A -85,B 0,C 180,E1 -8067.715,E2 -8067.715} C_VEL
LIN {X 0,Y 460.536,Z 99.428,A -85,B 0,C 180,E1 -8070.769,E2 -8070.769} C_VEL
LIN {X 0,Y 460.558,Z 99.427,A -85,B 0,C 180,E1 -8073.735,E2 -8073.735} C_VEL
LIN {X 0,Y 460.542,Z 99.427,A -85,B 0,C 180,E1 -8076.624,E2 -8076.624} C_VEL
LIN {X 0,Y 460.547,Z 99.427,A -85,B 0,C 180,E1 -8079.453,E2 -8079.453} C_VEL
LIN {X 0,Y 460.555,Z 99.428,A -85,B 0,C 180,E1 -8082.23,E2 -8082.23} C_VEL
LIN {X 0,Y 460.565,Z 99.423,A -85,B 0,C 180,E1 -8084.965,E2 -8084.965} C_VEL
LIN {X 0,Y 460.624,Z 99.421,A -85,B 0,C 180,E1 -8087.666,E2 -8087.666} C_VEL
LIN {X 0,Y 460.624,Z 99.417,A -85,B 0,C 180,E1 -8091.224,E2 -8091.224} C_VEL
LIN {X 0,Y 460.705,Z 99.412,A -85,B 0,C 180,E1 -8093.87,E2 -8093.87} C_VEL
LIN {X 0,Y 460.82,Z 99.395,A -85,B 0,C 180,E1 -8097.378,E2 -8097.378} C_VEL
LIN {X 0,Y 460.849,Z 99.391,A -85,B 0,C 180,E1 -8100,E2 -8100} C_VEL
LIN {X 0,Y 460.82,Z 99.391,A -85,B 0,C 180,E1 -8102.622,E2 -8102.622} C_VEL
LIN {X 0,Y 460.705,Z 99.407,A -85,B 0,C 180,E1 -8106.13,E2 -8106.13} C_VEL
LIN {X 0,Y 460.624,Z 99.416,A -85,B 0,C 180,E1 -8108.776,E2 -8108.776} C_VEL
LIN {X 0,Y 460.609,Z 99.417,A -85,B 0,C 180,E1 -8112.445,E2 -8112.445} C_VEL
LIN {X 0,Y 460.596,Z 99.42,A -85,B 0,C 180,E1 -8115.998,E2 -8115.998} C_VEL
LIN {X 0,Y 460.567,Z 99.426,A -85,B 0,C 180,E1 -8118.902,E2 -8118.902} C_VEL
LIN {X 0,Y 460.512,Z 99.435,A -85,B 0,C 180,E1 -8121.486,E2 -8121.486} C_VEL
LIN {X 0,Y 460.539,Z 99.426,A -85,B 0,C 180,E1 -8124.332,E2 -8124.332} C_VEL
LIN {X 0,Y 460.569,Z 99.429,A -85,B 0,C 180,E1 -8127.244,E2 -8127.244} C_VEL
LIN {X 0,Y 460.507,Z 99.43,A -85,B 0,C 180,E1 -8130.24,E2 -8130.24} C_VEL
LIN {X 0,Y 460.525,Z 99.432,A -85,B 0,C 180,E1 -8133.325,E2 -8133.325} C_VEL
LIN {X 0,Y 460.476,Z 99.436,A -85,B 0,C 180,E1 -8136.53,E2 -8136.53} C_VEL
LIN {X 0,Y 460.542,Z 99.433,A -85,B 0,C 180,E1 -8138.898,E2 -8138.898} C_VEL
LIN {X 0,Y 460.52,Z 99.429,A -85,B 0,C 180,E1 -8142.182,E2 -8142.182} C_VEL
LIN {X 0,Y 460.517,Z 99.43,A -85,B 0,C 180,E1 -8145.412,E2 -8145.412} C_VEL
LIN {X 0,Y 460.532,Z 99.43,A -85,B 0,C 180,E1 -8148.398,E2 -8148.398} C_VEL
LIN {X 0,Y 460.528,Z 99.429,A -85,B 0,C 180,E1 -8151.268,E2 -8151.268} C_VEL
LIN {X 0,Y 460.507,Z 99.437,A -85,B 0,C 180,E1 -8154.555,E2 -8154.555} C_VEL
LIN {X 0,Y 460.529,Z 99.427,A -85,B 0,C 180,E1 -8157.716,E2 -8157.716} C_VEL
LIN {X 0,Y 460.538,Z 99.432,A -85,B 0,C 180,E1 -8160.77,E2 -8160.77} C_VEL
LIN {X 0,Y 460.561,Z 99.424,A -85,B 0,C 180,E1 -8163.735,E2 -8163.735} C_VEL
LIN {X 0,Y 460.545,Z 99.431,A -85,B 0,C 180,E1 -8166.625,E2 -8166.625} C_VEL
LIN {X 0,Y 460.55,Z 99.425,A -85,B 0,C 180,E1 -8169.453,E2 -8169.453} C_VEL
LIN {X 0,Y 460.559,Z 99.43,A -85,B 0,C 180,E1 -8172.231,E2 -8172.231} C_VEL
LIN {X 0,Y 460.565,Z 99.424,A -85,B 0,C 180,E1 -8174.965,E2 -8174.965} C_VEL
LIN {X 0,Y 460.611,Z 99.421,A -85,B 0,C 180,E1 -8178.56,E2 -8178.56} C_VEL
LIN {X 0,Y 460.576,Z 99.422,A -85,B 0,C 180,E1 -8179.227,E2 -8179.227} C_VEL
LIN {X 0,Y 459.922,Z 99.51,A -85,B 0,C 180,E1 -8179.957,E2 -8179.957} C_VEL
LIN {X 0,Y 457.105,Z 99.855,A -85,B 0,C 180,E1 -8181.143,E2 -8181.143} C_VEL
LIN {X 0,Y 454.726,Z 100.157,A -85,B 0,C 180,E1 -8182.1,E2 -8182.1} C_VEL
LIN {X 0,Y 453.714,Z 100.278,A -85,B 0,C 180,E1 -8182.839,E2 -8182.839} C_VEL
LIN {X 0,Y 453.637,Z 100.286,A -85,B 0,C 180,E1 -8183.089,E2 -8183.089} C_VEL
LIN {X 0,Y 453.671,Z 100.284,A -85,B 0,C 180,E1 -8184.667,E2 -8184.667} C_VEL
LIN {X 0,Y 453.745,Z 100.273,A -85,B 0,C 180,E1 -8187.337,E2 -8187.337} C_VEL
LIN {X 0,Y 453.823,Z 100.27,A -85,B 0,C 180,E1 -8190.001,E2 -8190.001} C_VEL
LIN {X 0,Y 453.745,Z 100.274,A -85,B 0,C 180,E1 -8192.664,E2 -8192.664} C_VEL
LIN {X 0,Y 453.678,Z 100.285,A -85,B 0,C 180,E1 -8196.226,E2 -8196.226} C_VEL
LIN {X 0,Y 453.593,Z 100.291,A -85,B 0,C 180,E1 -8198.914,E2 -8198.914} C_VEL
LIN {X 0,Y 453.565,Z 100.296,A -85,B 0,C 180,E1 -8202.529,E2 -8202.529} C_VEL
LIN {X 0,Y 453.547,Z 100.3,A -85,B 0,C 180,E1 -8206.196,E2 -8206.196} C_VEL
LIN {X 0,Y 453.522,Z 100.301,A -85,B 0,C 180,E1 -8209.041,E2 -8209.041} C_VEL
LIN {X 0,Y 453.478,Z 100.312,A -85,B 0,C 180,E1 -8211.837,E2 -8211.837} C_VEL
LIN {X 0,Y 453.503,Z 100.303,A -85,B 0,C 180,E1 -8214.736,E2 -8214.736} C_VEL
LIN {X 0,Y 453.54,Z 100.301,A -85,B 0,C 180,E1 -8217.961,E2 -8217.961} C_VEL
LIN {X 0,Y 453.469,Z 100.315,A -85,B 0,C 180,E1 -8221.526,E2 -8221.526} C_VEL
LIN {X 0,Y 453.49,Z 100.305,A -85,B 0,C 180,E1 -8224.778,E2 -8224.778} C_VEL
LIN {X 0,Y 453.467,Z 100.307,A -85,B 0,C 180,E1 -8228.312,E2 -8228.312} C_VEL
LIN {X 0,Y 453.497,Z 100.304,A -85,B 0,C 180,E1 -8230.609,E2 -8230.609} C_VEL
LIN {X 0,Y 453.475,Z 100.306,A -85,B 0,C 180,E1 -8234.221,E2 -8234.221} C_VEL
LIN {X 0,Y 453.466,Z 100.312,A -85,B 0,C 180,E1 -8237.005,E2 -8237.005} C_VEL
LIN {X 0,Y 453.497,Z 100.309,A -85,B 0,C 180,E1 -8239.409,E2 -8239.409} C_VEL
LIN {X 0,Y 453.453,Z 100.309,A -85,B 0,C 180,E1 -8242.228,E2 -8242.228} C_VEL
LIN {X 0,Y 453.492,Z 100.311,A -85,B 0,C 180,E1 -8245.223,E2 -8245.223} C_VEL
LIN {X 0,Y 453.469,Z 100.312,A -85,B 0,C 180,E1 -8248.475,E2 -8248.475} C_VEL
LIN {X 0,Y 453.465,Z 100.312,A -85,B 0,C 180,E1 -8250.028,E2 -8250.028} C_VEL
LIN {X 0,Y 454.499,Z 103.192,A -85,B 0,C 180,E1 -8250.174,E2 -8250.174} C_VEL
LIN {X 0,Y 466.602,Z 127.255,A -85,B 0,C 180,E1 -8251.437,E2 -8251.437} C_VEL
LIN {X 0,Y 463.56,Z 260.236,A -85,B 0,C 180,E1 -8253.866,E2 -8253.866} C_VEL
LIN {X 0,Y 462.874,Z 294.575,A -85,B 0,C 180,E1 -8254.51,E2 -8254.51} C_VEL
LIN {X 0,Y 462.334,Z 311.173,A -85,B 0,C 180,E1 -8254.99,E2 -8254.99} C_VEL
LIN {X 0,Y 461.676,Z 326.832,A -85,B 0,C 180,E1 -8255.612,E2 -8255.612} C_VEL
LIN {X 0,Y 460.91,Z 341.367,A -85,B 0,C 180,E1 -8256.34,E2 -8256.34} C_VEL
LIN {X 0,Y 459.932,Z 357.021,A -85,B 0,C 180,E1 -8257.305,E2 -8257.305} C_VEL
LIN {X 0,Y 458.867,Z 372.066,A -85,B 0,C 180,E1 -8258.433,E2 -8258.433} C_VEL
LIN {X 0,Y 457.835,Z 386.032,A -85,B 0,C 180,E1 -8259.696,E2 -8259.696} C_VEL
LIN {X 0,Y 457,Z 397.561,A -85,B 0,C 180,E1 -8260.926,E2 -8260.926} C_VEL
LIN {X 0,Y 455.982,Z 410.311,A -85,B 0,C 180,E1 -8262.509,E2 -8262.509} C_VEL
LIN {X 0,Y 455.178,Z 421.119,A -85,B 0,C 180,E1 -8264.094,E2 -8264.094} C_VEL
LIN {X 0,Y 454.396,Z 431.517,A -85,B 0,C 180,E1 -8265.901,E2 -8265.901} C_VEL
LIN {X 0,Y 453.889,Z 439.149,A -85,B 0,C 180,E1 -8267.48,E2 -8267.48} C_VEL
LIN {X 0,Y 453.384,Z 446.493,A -85,B 0,C 180,E1 -8269.28,E2 -8269.28} C_VEL
LIN {X 0,Y 453.13,Z 452.549,A -85,B 0,C 180,E1 -8271.077,E2 -8271.077} C_VEL
LIN {X 0,Y 452.952,Z 458.203,A -85,B 0,C 180,E1 -8273.231,E2 -8273.231} C_VEL
LIN {X 0,Y 452.753,Z 462.512,A -85,B 0,C 180,E1 -8275.548,E2 -8275.548} C_VEL
LIN {X 0,Y 452.72,Z 464.61,A -85,B 0,C 180,E1 -8277.331,E2 -8277.331} C_VEL
LIN {X 0,Y 452.517,Z 465.784,A -85,B 0,C 180,E1 -8279.11,E2 -8279.11} C_VEL
LIN {X 0,Y 452.52,Z 465.927,A -85,B 0,C 180,E1 -8280.89,E2 -8280.89} C_VEL
LIN {X 0,Y 452.729,Z 465.083,A -85,B 0,C 180,E1 -8282.669,E2 -8282.669} C_VEL
LIN {X 0,Y 452.8,Z 463.262,A -85,B 0,C 180,E1 -8284.451,E2 -8284.451} C_VEL
LIN {X 0,Y 452.902,Z 460.391,A -85,B 0,C 180,E1 -8286.236,E2 -8286.236} C_VEL
LIN {X 0,Y 453.151,Z 456.499,A -85,B 0,C 180,E1 -8288.024,E2 -8288.024} C_VEL
LIN {X 0,Y 453.515,Z 449.976,A -85,B 0,C 180,E1 -8290.266,E2 -8290.266} C_VEL
LIN {X 0,Y 453.981,Z 443.297,A -85,B 0,C 180,E1 -8292.063,E2 -8292.063} C_VEL
LIN {X 0,Y 454.557,Z 435.208,A -85,B 0,C 180,E1 -8293.866,E2 -8293.866} C_VEL
LIN {X 0,Y 455.386,Z 425.473,A -85,B 0,C 180,E1 -8295.669,E2 -8295.669} C_VEL
LIN {X 0,Y 456.177,Z 415.642,A -85,B 0,C 180,E1 -8297.216,E2 -8297.216} C_VEL
LIN {X 0,Y 457.218,Z 403.454,A -85,B 0,C 180,E1 -8298.832,E2 -8298.832} C_VEL
LIN {X 0,Y 458.224,Z 390.323,A -85,B 0,C 180,E1 -8300.301,E2 -8300.301} C_VEL
LIN {X 0,Y 459.411,Z 375.711,A -85,B 0,C 180,E1 -8301.658,E2 -8301.658} C_VEL
LIN {X 0,Y 460.346,Z 362.634,A -85,B 0,C 180,E1 -8302.674,E2 -8302.674} C_VEL
LIN {X 0,Y 461.231,Z 349.053,A -85,B 0,C 180,E1 -8303.567,E2 -8303.567} C_VEL
LIN {X 0,Y 462.078,Z 334.404,A -85,B 0,C 180,E1 -8304.366,E2 -8304.366} C_VEL
LIN {X 0,Y 462.814,Z 317.175,A -85,B 0,C 180,E1 -8305.102,E2 -8305.102} C_VEL
LIN {X 0,Y 463.384,Z 299.947,A -85,B 0,C 180,E1 -8305.64,E2 -8305.64} C_VEL
LIN {X 0,Y 466.429,Z 206.758,A -85,B 0,C 180,E1 -8307.594,E2 -8307.594} C_VEL
LIN {X 0,Y 470.097,Z 129.873,A -85,B 0,C 180,E1 -8309.326,E2 -8309.326} C_VEL
LIN {X 0,Y 468.806,Z 126.708,A -85,B 0,C 180,E1 -8309.545,E2 -8309.545} C_VEL
LIN {X 0,Y 462.894,Z 115.972,A -85,B 0,C 180,E1 -8310.504,E2 -8310.504} C_VEL
LIN {X 0,Y 460.304,Z 111.877,A -85,B 0,C 180,E1 -8310.941,E2 -8310.941} C_VEL
LIN {X 0,Y 458.226,Z 108.578,A -85,B 0,C 180,E1 -8311.307,E2 -8311.307} C_VEL
LIN {X 0,Y 456.396,Z 105.336,A -85,B 0,C 180,E1 -8311.66,E2 -8311.66} C_VEL
LIN {X 0,Y 454.173,Z 102.553,A -85,B 0,C 180,E1 -8312.058,E2 -8312.058} C_VEL
LIN {X 0,Y 453.819,Z 101.728,A -85,B 0,C 180,E1 -8312.144,E2 -8312.144} C_VEL
LIN {X 0,Y 453.487,Z 100.313,A -85,B 0,C 180,E1 -8312.519,E2 -8312.519} C_VEL
LIN {X 0,Y 453.477,Z 100.313,A -85,B 0,C 180,E1 -8314.989,E2 -8314.989} C_VEL
LIN {X 0,Y 453.46,Z 100.316,A -85,B 0,C 180,E1 -8318.312,E2 -8318.312} C_VEL
LIN {X 0,Y 453.496,Z 100.31,A -85,B 0,C 180,E1 -8320.608,E2 -8320.608} C_VEL
LIN {X 0,Y 453.456,Z 100.314,A -85,B 0,C 180,E1 -8323.244,E2 -8323.244} C_VEL
LIN {X 0,Y 453.465,Z 100.315,A -85,B 0,C 180,E1 -8325.778,E2 -8325.778} C_VEL
LIN {X 0,Y 453.481,Z 100.313,A -85,B 0,C 180,E1 -8328.209,E2 -8328.209} C_VEL
LIN {X 0,Y 453.496,Z 100.31,A -85,B 0,C 180,E1 -8330.793,E2 -8330.793} C_VEL
LIN {X 0,Y 453.488,Z 100.414,A -85,B 0,C 180,E1 -8331.945,E2 -8331.945} C_VEL
LIN {X 0,Y 456.744,Z 108.349,A -85,B 0,C 180,E1 -8333.778,E2 -8333.778} C_VEL
LIN {X 0,Y 459.814,Z 116.192,A -85,B 0,C 180,E1 -8335.322,E2 -8335.322} C_VEL
LIN {X 0,Y 462.75,Z 125.198,A -85,B 0,C 180,E1 -8336.855,E2 -8336.855} C_VEL
LIN {X 0,Y 464.784,Z 133.207,A -85,B 0,C 180,E1 -8338.046,E2 -8338.046} C_VEL
LIN {X 0,Y 463.886,Z 142.466,A -85,B 0,C 180,E1 -8339.036,E2 -8339.036} C_VEL
LIN {X 0,Y 466.34,Z 159.437,A -85,B 0,C 180,E1 -8339.788,E2 -8339.788} C_VEL
LIN {X 0,Y 468.331,Z 176.913,A -85,B 0,C 180,E1 -8340.458,E2 -8340.458} C_VEL
LIN {X 0,Y 468.762,Z 183.181,A -85,B 0,C 180,E1 -8340.665,E2 -8340.665} C_VEL
LIN {X 0,Y 465.167,Z 269.081,A -85,B 0,C 180,E1 -8342.53,E2 -8342.53} C_VEL
LIN {X 0,Y 462.54,Z 357.993,A -85,B 0,C 180,E1 -8344.339,E2 -8344.339} C_VEL
LIN {X 0,Y 461.581,Z 375.478,A -85,B 0,C 180,E1 -8344.855,E2 -8344.855} C_VEL
LIN {X 0,Y 460.636,Z 392.645,A -85,B 0,C 180,E1 -8345.552,E2 -8345.552} C_VEL
LIN {X 0,Y 459.451,Z 409.824,A -85,B 0,C 180,E1 -8346.445,E2 -8346.445} C_VEL
LIN {X 0,Y 458.307,Z 425.519,A -85,B 0,C 180,E1 -8347.457,E2 -8347.457} C_VEL
LIN {X 0,Y 457.263,Z 440.124,A -85,B 0,C 180,E1 -8348.59,E2 -8348.59} C_VEL
LIN {X 0,Y 456.268,Z 454.36,A -85,B 0,C 180,E1 -8349.896,E2 -8349.896} C_VEL
LIN {X 0,Y 455.448,Z 465.646,A -85,B 0,C 180,E1 -8351.091,E2 -8351.091} C_VEL
LIN {X 0,Y 454.588,Z 478.485,A -85,B 0,C 180,E1 -8352.685,E2 -8352.685} C_VEL
LIN {X 0,Y 453.92,Z 489.392,A -85,B 0,C 180,E1 -8354.279,E2 -8354.279} C_VEL
LIN {X 0,Y 453.404,Z 499.978,A -85,B 0,C 180,E1 -8356.098,E2 -8356.098} C_VEL
LIN {X 0,Y 453.032,Z 508.852,A -85,B 0,C 180,E1 -8357.915,E2 -8357.915} C_VEL
LIN {X 0,Y 452.763,Z 516.198,A -85,B 0,C 180,E1 -8359.717,E2 -8359.717} C_VEL
LIN {X 0,Y 452.668,Z 523.465,A -85,B 0,C 180,E1 -8361.967,E2 -8361.967} C_VEL
LIN {X 0,Y 452.65,Z 527.855,A -85,B 0,C 180,E1 -8363.76,E2 -8363.76} C_VEL
LIN {X 0,Y 452.54,Z 531.153,A -85,B 0,C 180,E1 -8365.546,E2 -8365.546} C_VEL
LIN {X 0,Y 452.644,Z 533.339,A -85,B 0,C 180,E1 -8367.33,E2 -8367.33} C_VEL
LIN {X 0,Y 452.499,Z 534.454,A -85,B 0,C 180,E1 -8369.109,E2 -8369.109} C_VEL
LIN {X 0,Y 452.498,Z 534.539,A -85,B 0,C 180,E1 -8370.889,E2 -8370.889} C_VEL
LIN {X 0,Y 452.626,Z 533.56,A -85,B 0,C 180,E1 -8372.669,E2 -8372.669} C_VEL
LIN {X 0,Y 452.519,Z 531.55,A -85,B 0,C 180,E1 -8374.453,E2 -8374.453} C_VEL
LIN {X 0,Y 452.646,Z 527.999,A -85,B 0,C 180,E1 -8376.44,E2 -8376.44} C_VEL
LIN {X 0,Y 452.671,Z 522.925,A -85,B 0,C 180,E1 -8378.481,E2 -8378.481} C_VEL
LIN {X 0,Y 452.76,Z 517.207,A -85,B 0,C 180,E1 -8380.282,E2 -8380.282} C_VEL
LIN {X 0,Y 453.122,Z 509.328,A -85,B 0,C 180,E1 -8382.276,E2 -8382.276} C_VEL
LIN {X 0,Y 453.496,Z 500.367,A -85,B 0,C 180,E1 -8384.127,E2 -8384.127} C_VEL
LIN {X 0,Y 454.019,Z 491.264,A -85,B 0,C 180,E1 -8385.717,E2 -8385.717} C_VEL
LIN {X 0,Y 454.762,Z 480.668,A -85,B 0,C 180,E1 -8387.306,E2 -8387.306} C_VEL
LIN {X 0,Y 455.5,Z 470.083,A -85,B 0,C 180,E1 -8388.672,E2 -8388.672} C_VEL
LIN {X 0,Y 456.519,Z 457.115,A -85,B 0,C 180,E1 -8390.103,E2 -8390.103} C_VEL
LIN {X 0,Y 457.557,Z 443.343,A -85,B 0,C 180,E1 -8391.394,E2 -8391.394} C_VEL
LIN {X 0,Y 458.629,Z 429.031,A -85,B 0,C 180,E1 -8392.525,E2 -8392.525} C_VEL
LIN {X 0,Y 459.728,Z 413.935,A -85,B 0,C 180,E1 -8393.516,E2 -8393.516} C_VEL
LIN {X 0,Y 460.694,Z 398.766,A -85,B 0,C 180,E1 -8394.323,E2 -8394.323} C_VEL
LIN {X 0,Y 461.636,Z 382.099,A -85,B 0,C 180,E1 -8395.02,E2 -8395.02} C_VEL
LIN {X 0,Y 462.36,Z 366.029,A -85,B 0,C 180,E1 -8395.52,E2 -8395.52} C_VEL
LIN {X 0,Y 462.961,Z 347.646,A -85,B 0,C 180,E1 -8395.906,E2 -8395.906} C_VEL
LIN {X 0,Y 466.726,Z 181.325,A -85,B 0,C 180,E1 -8398.933,E2 -8398.933} C_VEL
LIN {X 0,Y 462.442,Z 152.049,A -85,B 0,C 180,E1 -8399.802,E2 -8399.802} C_VEL
LIN {X 0,Y 463.68,Z 132.46,A -85,B 0,C 180,E1 -8401.696,E2 -8401.696} C_VEL
LIN {X 0,Y 458.989,Z 117.004,A -85,B 0,C 180,E1 -8403.597,E2 -8403.597} C_VEL
LIN {X 0,Y 453.484,Z 100.311,A -85,B 0,C 180,E1 -8405.773,E2 -8405.773} C_VEL
LIN {X 0,Y 453.485,Z 100.309,A -85,B 0,C 180,E1 -8409.449,E2 -8409.449} C_VEL
LIN {X 0,Y 453.488,Z 100.308,A -85,B 0,C 180,E1 -8412.991,E2 -8412.991} C_VEL
LIN {X 0,Y 453.462,Z 100.312,A -85,B 0,C 180,E1 -8415.779,E2 -8415.779} C_VEL
LIN {X 0,Y 453.474,Z 100.312,A -85,B 0,C 180,E1 -8418.209,E2 -8418.209} C_VEL
LIN {X 0,Y 453.511,Z 100.304,A -85,B 0,C 180,E1 -8420.79,E2 -8420.79} C_VEL
LIN {X 0,Y 453.452,Z 100.313,A -85,B 0,C 180,E1 -8423.917,E2 -8423.917} C_VEL
LIN {X 0,Y 453.478,Z 100.306,A -85,B 0,C 180,E1 -8427.151,E2 -8427.151} C_VEL
LIN {X 0,Y 453.509,Z 100.308,A -85,B 0,C 180,E1 -8430.271,E2 -8430.271} C_VEL
LIN {X 0,Y 453.504,Z 100.303,A -85,B 0,C 180,E1 -8433.294,E2 -8433.294} C_VEL
LIN {X 0,Y 453.499,Z 100.309,A -85,B 0,C 180,E1 -8436.239,E2 -8436.239} C_VEL
LIN {X 0,Y 453.478,Z 100.306,A -85,B 0,C 180,E1 -8439.118,E2 -8439.118} C_VEL
LIN {X 0,Y 453.508,Z 100.31,A -85,B 0,C 180,E1 -8441.945,E2 -8441.945} C_VEL
LIN {X 0,Y 453.545,Z 100.298,A -85,B 0,C 180,E1 -8444.727,E2 -8444.727} C_VEL
LIN {X 0,Y 453.597,Z 100.294,A -85,B 0,C 180,E1 -8447.472,E2 -8447.472} C_VEL
LIN {X 0,Y 453.588,Z 100.293,A -85,B 0,C 180,E1 -8451.087,E2 -8451.087} C_VEL
LIN {X 0,Y 453.673,Z 100.289,A -85,B 0,C 180,E1 -8453.775,E2 -8453.775} C_VEL
LIN {X 0,Y 453.76,Z 100.274,A -85,B 0,C 180,E1 -8457.337,E2 -8457.337} C_VEL
LIN {X 0,Y 453.819,Z 100.267,A -85,B 0,C 180,E1 -8460,E2 -8460} C_VEL
LIN {X 0,Y 453.761,Z 100.271,A -85,B 0,C 180,E1 -8462.663,E2 -8462.663} C_VEL
LIN {X 0,Y 453.673,Z 100.282,A -85,B 0,C 180,E1 -8466.225,E2 -8466.225} C_VEL
LIN {X 0,Y 453.587,Z 100.294,A -85,B 0,C 180,E1 -8468.914,E2 -8468.914} C_VEL
LIN {X 0,Y 453.559,Z 100.296,A -85,B 0,C 180,E1 -8472.529,E2 -8472.529} C_VEL
LIN {X 0,Y 453.54,Z 100.298,A -85,B 0,C 180,E1 -8476.196,E2 -8476.196} C_VEL
LIN {X 0,Y 453.517,Z 100.306,A -85,B 0,C 180,E1 -8479.041,E2 -8479.041} C_VEL
LIN {X 0,Y 453.473,Z 100.308,A -85,B 0,C 180,E1 -8481.836,E2 -8481.836} C_VEL
LIN {X 0,Y 453.51,Z 100.304,A -85,B 0,C 180,E1 -8484.735,E2 -8484.735} C_VEL
LIN {X 0,Y 453.528,Z 100.3,A -85,B 0,C 180,E1 -8487.96,E2 -8487.96} C_VEL
LIN {X 0,Y 453.463,Z 100.31,A -85,B 0,C 180,E1 -8491.526,E2 -8491.526} C_VEL
LIN {X 0,Y 453.485,Z 100.31,A -85,B 0,C 180,E1 -8494.778,E2 -8494.778} C_VEL
LIN {X 0,Y 453.47,Z 100.308,A -85,B 0,C 180,E1 -8498.311,E2 -8498.311} C_VEL
LIN {X 0,Y 453.49,Z 100.308,A -85,B 0,C 180,E1 -8500.609,E2 -8500.609} C_VEL
LIN {X 0,Y 453.461,Z 100.311,A -85,B 0,C 180,E1 -8503.246,E2 -8503.246} C_VEL
LIN {X 0,Y 453.47,Z 100.307,A -85,B 0,C 180,E1 -8505.78,E2 -8505.78} C_VEL
LIN {X 0,Y 453.512,Z 100.303,A -85,B 0,C 180,E1 -8509.406,E2 -8509.406} C_VEL
LIN {X 0,Y 453.447,Z 100.312,A -85,B 0,C 180,E1 -8512.228,E2 -8512.228} C_VEL
LIN {X 0,Y 453.484,Z 100.307,A -85,B 0,C 180,E1 -8515.223,E2 -8515.223} C_VEL
LIN {X 0,Y 453.464,Z 100.314,A -85,B 0,C 180,E1 -8518.475,E2 -8518.475} C_VEL
LIN {X 0,Y 453.535,Z 100.301,A -85,B 0,C 180,E1 -8522.04,E2 -8522.04} C_VEL
LIN {X 0,Y 453.512,Z 100.302,A -85,B 0,C 180,E1 -8525.266,E2 -8525.266} C_VEL
LIN {X 0,Y 453.479,Z 100.314,A -85,B 0,C 180,E1 -8528.416,E2 -8528.416} C_VEL
LIN {X 0,Y 453.521,Z 100.302,A -85,B 0,C 180,E1 -8531.009,E2 -8531.009} C_VEL
LIN {X 0,Y 453.568,Z 100.297,A -85,B 0,C 180,E1 -8533.88,E2 -8533.88} C_VEL
LIN {X 0,Y 453.563,Z 100.295,A -85,B 0,C 180,E1 -8537.472,E2 -8537.472} C_VEL
LIN {X 0,Y 453.592,Z 100.292,A -85,B 0,C 180,E1 -8541.087,E2 -8541.087} C_VEL
LIN {X 0,Y 453.637,Z 100.286,A -85,B 0,C 180,E1 -8543.089,E2 -8543.089} C_VEL
LIN {X 0,Y 452.952,Z 100.377,A -85,B 0,C 180,E1 -8543.83,E2 -8543.83} C_VEL
LIN {X 0,Y 450.005,Z 100.74,A -85,B 0,C 180,E1 -8545.032,E2 -8545.032} C_VEL
LIN {X 0,Y 447.579,Z 101.047,A -85,B 0,C 180,E1 -8546.001,E2 -8546.001} C_VEL
LIN {X 0,Y 446.635,Z 101.16,A -85,B 0,C 180,E1 -8546.751,E2 -8546.751} C_VEL
LIN {X 0,Y 446.611,Z 101.161,A -85,B 0,C 180,E1 -8547.005,E2 -8547.005} C_VEL
LIN {X 0,Y 446.793,Z 101.146,A -85,B 0,C 180,E1 -8550.001,E2 -8550.001} C_VEL
LIN {X 0,Y 446.692,Z 101.152,A -85,B 0,C 180,E1 -8552.706,E2 -8552.706} C_VEL
LIN {X 0,Y 446.647,Z 101.16,A -85,B 0,C 180,E1 -8556.324,E2 -8556.324} C_VEL
LIN {X 0,Y 446.539,Z 101.17,A -85,B 0,C 180,E1 -8559.056,E2 -8559.056} C_VEL
LIN {X 0,Y 446.523,Z 101.172,A -85,B 0,C 180,E1 -8562.73,E2 -8562.73} C_VEL
LIN {X 0,Y 446.498,Z 101.178,A -85,B 0,C 180,E1 -8566.228,E2 -8566.228} C_VEL
LIN {X 0,Y 446.471,Z 101.181,A -85,B 0,C 180,E1 -8569.304,E2 -8569.304} C_VEL
LIN {X 0,Y 446.42,Z 101.187,A -85,B 0,C 180,E1 -8572.2,E2 -8572.2} C_VEL
LIN {X 0,Y 446.446,Z 101.184,A -85,B 0,C 180,E1 -8575.154,E2 -8575.154} C_VEL
LIN {X 0,Y 446.487,Z 101.178,A -85,B 0,C 180,E1 -8578.179,E2 -8578.179} C_VEL
LIN {X 0,Y 446.422,Z 101.189,A -85,B 0,C 180,E1 -8581.775,E2 -8581.775} C_VEL
LIN {X 0,Y 446.431,Z 101.184,A -85,B 0,C 180,E1 -8584.523,E2 -8584.523} C_VEL
LIN {X 0,Y 446.418,Z 101.186,A -85,B 0,C 180,E1 -8588.08,E2 -8588.08} C_VEL
LIN {X 0,Y 446.43,Z 101.186,A -85,B 0,C 180,E1 -8590.918,E2 -8590.918} C_VEL
LIN {X 0,Y 446.425,Z 101.186,A -85,B 0,C 180,E1 -8593.844,E2 -8593.844} C_VEL
LIN {X 0,Y 446.402,Z 101.187,A -85,B 0,C 180,E1 -8596.404,E2 -8596.404} C_VEL
LIN {X 0,Y 446.43,Z 101.19,A -85,B 0,C 180,E1 -8599.083,E2 -8599.083} C_VEL
LIN {X 0,Y 446.412,Z 101.186,A -85,B 0,C 180,E1 -8602.122,E2 -8602.122} C_VEL
LIN {X 0,Y 446.433,Z 101.188,A -85,B 0,C 180,E1 -8605.477,E2 -8605.477} C_VEL
LIN {X 0,Y 446.42,Z 101.19,A -85,B 0,C 180,E1 -8608.7,E2 -8608.7} C_VEL
LIN {X 0,Y 446.432,Z 101.188,A -85,B 0,C 180,E1 -8609.58,E2 -8609.58} C_VEL
LIN {X 0,Y 447.536,Z 104.205,A -85,B 0,C 180,E1 -8609.736,E2 -8609.736} C_VEL
LIN {X 0,Y 460.229,Z 129.449,A -85,B 0,C 180,E1 -8611.089,E2 -8611.089} C_VEL
LIN {X 0,Y 456.68,Z 277.03,A -85,B 0,C 180,E1 -8613.832,E2 -8613.832} C_VEL
LIN {X 0,Y 456.184,Z 297.684,A -85,B 0,C 180,E1 -8614.262,E2 -8614.262} C_VEL
LIN {X 0,Y 455.586,Z 314.298,A -85,B 0,C 180,E1 -8614.776,E2 -8614.776} C_VEL
LIN {X 0,Y 454.847,Z 330.31,A -85,B 0,C 180,E1 -8615.446,E2 -8615.446} C_VEL
LIN {X 0,Y 454.047,Z 345.599,A -85,B 0,C 180,E1 -8616.269,E2 -8616.269} C_VEL
LIN {X 0,Y 452.935,Z 361.233,A -85,B 0,C 180,E1 -8617.296,E2 -8617.296} C_VEL
LIN {X 0,Y 451.879,Z 375.625,A -85,B 0,C 180,E1 -8618.442,E2 -8618.442} C_VEL
LIN {X 0,Y 450.82,Z 389.458,A -85,B 0,C 180,E1 -8619.757,E2 -8619.757} C_VEL
LIN {X 0,Y 449.85,Z 401.382,A -85,B 0,C 180,E1 -8621.084,E2 -8621.084} C_VEL
LIN {X 0,Y 448.816,Z 414.271,A -85,B 0,C 180,E1 -8622.786,E2 -8622.786} C_VEL
LIN {X 0,Y 447.947,Z 425.347,A -85,B 0,C 180,E1 -8624.531,E2 -8624.531} C_VEL
LIN {X 0,Y 447.227,Z 435.117,A -85,B 0,C 180,E1 -8626.366,E2 -8626.366} C_VEL
LIN {X 0,Y 446.666,Z 443.257,A -85,B 0,C 180,E1 -8628.197,E2 -8628.197} C_VEL
LIN {X 0,Y 446.232,Z 450.01,A -85,B 0,C 180,E1 -8630.023,E2 -8630.023} C_VEL
LIN {X 0,Y 445.988,Z 455.478,A -85,B 0,C 180,E1 -8631.846,E2 -8631.846} C_VEL
LIN {X 0,Y 445.83,Z 459.74,A -85,B 0,C 180,E1 -8633.665,E2 -8633.665} C_VEL
LIN {X 0,Y 445.684,Z 462.993,A -85,B 0,C 180,E1 -8635.478,E2 -8635.478} C_VEL
LIN {X 0,Y 445.668,Z 465.115,A -85,B 0,C 180,E1 -8637.288,E2 -8637.288} C_VEL
LIN {X 0,Y 445.453,Z 466.327,A -85,B 0,C 180,E1 -8639.096,E2 -8639.096} C_VEL
LIN {X 0,Y 445.456,Z 466.489,A -85,B 0,C 180,E1 -8640.904,E2 -8640.904} C_VEL
LIN {X 0,Y 445.68,Z 465.667,A -85,B 0,C 180,E1 -8642.711,E2 -8642.711} C_VEL
LIN {X 0,Y 445.749,Z 463.859,A -85,B 0,C 180,E1 -8644.521,E2 -8644.521} C_VEL
LIN {X 0,Y 445.87,Z 461.004,A -85,B 0,C 180,E1 -8646.335,E2 -8646.335} C_VEL
LIN {X 0,Y 446.124,Z 457.126,A -85,B 0,C 180,E1 -8648.151,E2 -8648.151} C_VEL
LIN {X 0,Y 446.545,Z 450.609,A -85,B 0,C 180,E1 -8650.428,E2 -8650.428} C_VEL
LIN {X 0,Y 447.034,Z 443.943,A -85,B 0,C 180,E1 -8652.253,E2 -8652.253} C_VEL
LIN {X 0,Y 447.667,Z 435.857,A -85,B 0,C 180,E1 -8654.083,E2 -8654.083} C_VEL
LIN {X 0,Y 448.555,Z 426.138,A -85,B 0,C 180,E1 -8655.914,E2 -8655.914} C_VEL
LIN {X 0,Y 449.47,Z 415.537,A -85,B 0,C 180,E1 -8657.594,E2 -8657.594} C_VEL
LIN {X 0,Y 450.509,Z 404.146,A -85,B 0,C 180,E1 -8659.123,E2 -8659.123} C_VEL
LIN {X 0,Y 451.588,Z 391.173,A -85,B 0,C 180,E1 -8660.597,E2 -8660.597} C_VEL
LIN {X 0,Y 452.748,Z 377.741,A -85,B 0,C 180,E1 -8661.873,E2 -8661.873} C_VEL
LIN {X 0,Y 453.843,Z 363.448,A -85,B 0,C 180,E1 -8663.017,E2 -8663.017} C_VEL
LIN {X 0,Y 454.772,Z 350.105,A -85,B 0,C 180,E1 -8663.913,E2 -8663.913} C_VEL
LIN {X 0,Y 455.686,Z 335.43,A -85,B 0,C 180,E1 -8664.73,E2 -8664.73} C_VEL
LIN {X 0,Y 456.478,Z 318.457,A -85,B 0,C 180,E1 -8665.476,E2 -8665.476} C_VEL
LIN {X 0,Y 457.106,Z 301.627,A -85,B 0,C 180,E1 -8666.019,E2 -8666.019} C_VEL
LIN {X 0,Y 457.957,Z 274.156,A -85,B 0,C 180,E1 -8666.621,E2 -8666.621} C_VEL
LIN {X 0,Y 460.92,Z 199.885,A -85,B 0,C 180,E1 -8668.239,E2 -8668.239} C_VEL
LIN {X 0,Y 464.446,Z 131.853,A -85,B 0,C 180,E1 -8669.841,E2 -8669.841} C_VEL
LIN {X 0,Y 458.608,Z 120.945,A -85,B 0,C 180,E1 -8670.84,E2 -8670.84} C_VEL
LIN {X 0,Y 454.114,Z 113.682,A -85,B 0,C 180,E1 -8671.657,E2 -8671.657} C_VEL
LIN {X 0,Y 451.665,Z 109.845,A -85,B 0,C 180,E1 -8672.129,E2 -8672.129} C_VEL
LIN {X 0,Y 448.882,Z 105.708,A -85,B 0,C 180,E1 -8672.696,E2 -8672.696} C_VEL
LIN {X 0,Y 447.092,Z 103.341,A -85,B 0,C 180,E1 -8673.097,E2 -8673.097} C_VEL
LIN {X 0,Y 446.433,Z 101.19,A -85,B 0,C 180,E1 -8673.773,E2 -8673.773} C_VEL
LIN {X 0,Y 446.402,Z 101.194,A -85,B 0,C 180,E1 -8676.745,E2 -8676.745} C_VEL
LIN {X 0,Y 446.438,Z 101.19,A -85,B 0,C 180,E1 -8680.198,E2 -8680.198} C_VEL
LIN {X 0,Y 446.431,Z 101.19,A -85,B 0,C 180,E1 -8682.604,E2 -8682.604} C_VEL
LIN {X 0,Y 446.453,Z 101.186,A -85,B 0,C 180,E1 -8685.103,E2 -8685.103} C_VEL
LIN {X 0,Y 446.43,Z 101.19,A -85,B 0,C 180,E1 -8688.608,E2 -8688.608} C_VEL
LIN {X 0,Y 446.485,Z 101.319,A -85,B 0,C 180,E1 -8690.757,E2 -8690.757} C_VEL
LIN {X 0,Y 447.079,Z 103.408,A -85,B 0,C 180,E1 -8691.301,E2 -8691.301} C_VEL
LIN {X 0,Y 448.352,Z 105.986,A -85,B 0,C 180,E1 -8692.034,E2 -8692.034} C_VEL
LIN {X 0,Y 451.832,Z 114.241,A -85,B 0,C 180,E1 -8693.982,E2 -8693.982} C_VEL
LIN {X 0,Y 455.354,Z 123.827,A -85,B 0,C 180,E1 -8695.836,E2 -8695.836} C_VEL
LIN {X 0,Y 458.32,Z 134.327,A -85,B 0,C 180,E1 -8697.54,E2 -8697.54} C_VEL
LIN {X 0,Y 458.454,Z 137.075,A -85,B 0,C 180,E1 -8697.894,E2 -8697.894} C_VEL
LIN {X 0,Y 457.974,Z 141.257,A -85,B 0,C 180,E1 -8698.346,E2 -8698.346} C_VEL
LIN {X 0,Y 460.531,Z 158.45,A -85,B 0,C 180,E1 -8699.168,E2 -8699.168} C_VEL
LIN {X 0,Y 462.653,Z 178.66,A -85,B 0,C 180,E1 -8699.981,E2 -8699.981} C_VEL
LIN {X 0,Y 462.985,Z 184.134,A -85,B 0,C 180,E1 -8700.167,E2 -8700.167} C_VEL
LIN {X 0,Y 459.05,Z 270.24,A -85,B 0,C 180,E1 -8702.101,E2 -8702.101} C_VEL
LIN {X 0,Y 456.206,Z 356.995,A -85,B 0,C 180,E1 -8703.925,E2 -8703.925} C_VEL
LIN {X 0,Y 455.146,Z 375.109,A -85,B 0,C 180,E1 -8704.474,E2 -8704.474} C_VEL
LIN {X 0,Y 454.146,Z 392.068,A -85,B 0,C 180,E1 -8705.18,E2 -8705.18} C_VEL
LIN {X 0,Y 452.87,Z 409.146,A -85,B 0,C 180,E1 -8706.081,E2 -8706.081} C_VEL
LIN {X 0,Y 451.52,Z 426.409,A -85,B 0,C 180,E1 -8707.22,E2 -8707.22} C_VEL
LIN {X 0,Y 450.36,Z 442.087,A -85,B 0,C 180,E1 -8708.486,E2 -8708.486} C_VEL
LIN {X 0,Y 449.215,Z 456.457,A -85,B 0,C 180,E1 -8709.867,E2 -8709.867} C_VEL
LIN {X 0,Y 448.275,Z 468.726,A -85,B 0,C 180,E1 -8711.252,E2 -8711.252} C_VEL
LIN {X 0,Y 447.441,Z 481.027,A -85,B 0,C 180,E1 -8712.872,E2 -8712.872} C_VEL
LIN {X 0,Y 446.808,Z 491.559,A -85,B 0,C 180,E1 -8714.49,E2 -8714.49} C_VEL
LIN {X 0,Y 446.24,Z 501.711,A -85,B 0,C 180,E1 -8716.335,E2 -8716.335} C_VEL
LIN {X 0,Y 445.898,Z 510.15,A -85,B 0,C 180,E1 -8718.176,E2 -8718.176} C_VEL
LIN {X 0,Y 445.608,Z 517.137,A -85,B 0,C 180,E1 -8720.009,E2 -8720.009} C_VEL
LIN {X 0,Y 445.581,Z 522.867,A -85,B 0,C 180,E1 -8721.838,E2 -8721.838} C_VEL
LIN {X 0,Y 445.595,Z 527.278,A -85,B 0,C 180,E1 -8723.661,E2 -8723.661} C_VEL
LIN {X 0,Y 445.457,Z 530.589,A -85,B 0,C 180,E1 -8725.475,E2 -8725.475} C_VEL
LIN {X 0,Y 445.563,Z 532.791,A -85,B 0,C 180,E1 -8727.287,E2 -8727.287} C_VEL
LIN {X 0,Y 445.437,Z 533.908,A -85,B 0,C 180,E1 -8729.095,E2 -8729.095} C_VEL
LIN {X 0,Y 445.435,Z 533.996,A -85,B 0,C 180,E1 -8730.903,E2 -8730.903} C_VEL
LIN {X 0,Y 445.545,Z 533.004,A -85,B 0,C 180,E1 -8732.712,E2 -8732.712} C_VEL
LIN {X 0,Y 445.437,Z 530.985,A -85,B 0,C 180,E1 -8734.524,E2 -8734.524} C_VEL
LIN {X 0,Y 445.574,Z 527.616,A -85,B 0,C 180,E1 -8736.44,E2 -8736.44} C_VEL
LIN {X 0,Y 445.565,Z 523.584,A -85,B 0,C 180,E1 -8738.161,E2 -8738.161} C_VEL
LIN {X 0,Y 445.605,Z 518.07,A -85,B 0,C 180,E1 -8739.99,E2 -8739.99} C_VEL
LIN {X 0,Y 445.923,Z 511.285,A -85,B 0,C 180,E1 -8741.822,E2 -8741.822} C_VEL
LIN {X 0,Y 446.28,Z 503.075,A -85,B 0,C 180,E1 -8743.663,E2 -8743.663} C_VEL
LIN {X 0,Y 446.91,Z 493.232,A -85,B 0,C 180,E1 -8745.505,E2 -8745.505} C_VEL
LIN {X 0,Y 447.564,Z 483.065,A -85,B 0,C 180,E1 -8747.107,E2 -8747.107} C_VEL
LIN {X 0,Y 448.453,Z 470.917,A -85,B 0,C 180,E1 -8748.739,E2 -8748.739} C_VEL
LIN {X 0,Y 449.451,Z 458.859,A -85,B 0,C 180,E1 -8750.121,E2 -8750.121} C_VEL
LIN {X 0,Y 450.49,Z 446.016,A -85,B 0,C 180,E1 -8751.386,E2 -8751.386} C_VEL
LIN {X 0,Y 451.648,Z 430.719,A -85,B 0,C 180,E1 -8752.651,E2 -8752.651} C_VEL
LIN {X 0,Y 452.854,Z 415.191,A -85,B 0,C 180,E1 -8753.703,E2 -8753.703} C_VEL
LIN {X 0,Y 453.864,Z 400.266,A -85,B 0,C 180,E1 -8754.53,E2 -8754.53} C_VEL
LIN {X 0,Y 454.886,Z 383.534,A -85,B 0,C 180,E1 -8755.264,E2 -8755.264} C_VEL
LIN {X 0,Y 455.64,Z 367.269,A -85,B 0,C 180,E1 -8755.801,E2 -8755.801} C_VEL
LIN {X 0,Y 456.315,Z 349.853,A -85,B 0,C 180,E1 -8756.19,E2 -8756.19} C_VEL
LIN {X 0,Y 460.33,Z 182.219,A -85,B 0,C 180,E1 -8759.307,E2 -8759.307} C_VEL
LIN {X 0,Y 455.928,Z 151.544,A -85,B 0,C 180,E1 -8760.24,E2 -8760.24} C_VEL
LIN {X 0,Y 456.998,Z 135.392,A -85,B 0,C 180,E1 -8761.826,E2 -8761.826} C_VEL
LIN {X 0,Y 456.912,Z 133.596,A -85,B 0,C 180,E1 -8762.016,E2 -8762.016} C_VEL
LIN {X 0,Y 450.392,Z 113.159,A -85,B 0,C 180,E1 -8764.602,E2 -8764.602} C_VEL
LIN {X 0,Y 446.406,Z 101.194,A -85,B 0,C 180,E1 -8766.218,E2 -8766.218} C_VEL
LIN {X 0,Y 446.451,Z 101.186,A -85,B 0,C 180,E1 -8769.525,E2 -8769.525} C_VEL
LIN {X 0,Y 446.445,Z 101.19,A -85,B 0,C 180,E1 -8772.602,E2 -8772.602} C_VEL
LIN {X 0,Y 446.451,Z 101.185,A -85,B 0,C 180,E1 -8775.103,E2 -8775.103} C_VEL
LIN {X 0,Y 446.423,Z 101.189,A -85,B 0,C 180,E1 -8778.609,E2 -8778.609} C_VEL
LIN {X 0,Y 446.456,Z 101.181,A -85,B 0,C 180,E1 -8780.975,E2 -8780.975} C_VEL
LIN {X 0,Y 446.417,Z 101.192,A -85,B 0,C 180,E1 -8784.374,E2 -8784.374} C_VEL
LIN {X 0,Y 446.424,Z 101.186,A -85,B 0,C 180,E1 -8787.639,E2 -8787.639} C_VEL
LIN {X 0,Y 446.463,Z 101.181,A -85,B 0,C 180,E1 -8790.792,E2 -8790.792} C_VEL
LIN {X 0,Y 446.473,Z 101.183,A -85,B 0,C 180,E1 -8793.848,E2 -8793.848} C_VEL
LIN {X 0,Y 446.425,Z 101.185,A -85,B 0,C 180,E1 -8796.823,E2 -8796.823} C_VEL
LIN {X 0,Y 446.439,Z 101.187,A -85,B 0,C 180,E1 -8799.737,E2 -8799.737} C_VEL
LIN {X 0,Y 446.46,Z 101.181,A -85,B 0,C 180,E1 -8802.597,E2 -8802.597} C_VEL
LIN {X 0,Y 446.469,Z 101.181,A -85,B 0,C 180,E1 -8805.412,E2 -8805.412} C_VEL
LIN {X 0,Y 446.535,Z 101.174,A -85,B 0,C 180,E1 -8808.194,E2 -8808.194} C_VEL
LIN {X 0,Y 446.596,Z 101.17,A -85,B 0,C 180,E1 -8811.858,E2 -8811.858} C_VEL
LIN {X 0,Y 446.641,Z 101.158,A -85,B 0,C 180,E1 -8814.583,E2 -8814.583} C_VEL
LIN {X 0,Y 446.704,Z 101.153,A -85,B 0,C 180,E1 -8817.295,E2 -8817.295} C_VEL
LIN {X 0,Y 446.79,Z 101.142,A -85,B 0,C 180,E1 -8820,E2 -8820} C_VEL
LIN {X 0,Y 446.705,Z 101.15,A -85,B 0,C 180,E1 -8822.705,E2 -8822.705} C_VEL
LIN {X 0,Y 446.642,Z 101.158,A -85,B 0,C 180,E1 -8826.324,E2 -8826.324} C_VEL
LIN {X 0,Y 446.533,Z 101.174,A -85,B 0,C 180,E1 -8829.056,E2 -8829.056} C_VEL
LIN {X 0,Y 446.517,Z 101.174,A -85,B 0,C 180,E1 -8832.73,E2 -8832.73} C_VEL
LIN {X 0,Y 446.492,Z 101.176,A -85,B 0,C 180,E1 -8836.228,E2 -8836.228} C_VEL
LIN {X 0,Y 446.465,Z 101.187,A -85,B 0,C 180,E1 -8839.303,E2 -8839.303} C_VEL
LIN {X 0,Y 446.414,Z 101.186,A -85,B 0,C 180,E1 -8842.2,E2 -8842.2} C_VEL
LIN {X 0,Y 446.454,Z 101.188,A -85,B 0,C 180,E1 -8845.153,E2 -8845.153} C_VEL
LIN {X 0,Y 446.48,Z 101.178,A -85,B 0,C 180,E1 -8848.179,E2 -8848.179} C_VEL
LIN {X 0,Y 446.416,Z 101.186,A -85,B 0,C 180,E1 -8851.776,E2 -8851.776} C_VEL
LIN {X 0,Y 446.426,Z 101.186,A -85,B 0,C 180,E1 -8854.523,E2 -8854.523} C_VEL
LIN {X 0,Y 446.427,Z 101.184,A -85,B 0,C 180,E1 -8858.082,E2 -8858.082} C_VEL
LIN {X 0,Y 446.425,Z 101.193,A -85,B 0,C 180,E1 -8860.918,E2 -8860.918} C_VEL
LIN {X 0,Y 446.42,Z 101.185,A -85,B 0,C 180,E1 -8863.844,E2 -8863.844} C_VEL
LIN {X 0,Y 446.418,Z 101.188,A -85,B 0,C 180,E1 -8866.401,E2 -8866.401} C_VEL
LIN {X 0,Y 446.462,Z 101.18,A -85,B 0,C 180,E1 -8869.805,E2 -8869.805} C_VEL
LIN {X 0,Y 446.407,Z 101.188,A -85,B 0,C 180,E1 -8872.122,E2 -8872.122} C_VEL
LIN {X 0,Y 446.426,Z 101.185,A -85,B 0,C 180,E1 -8875.478,E2 -8875.478} C_VEL
LIN {X 0,Y 446.414,Z 101.192,A -85,B 0,C 180,E1 -8878.7,E2 -8878.7} C_VEL
LIN {X 0,Y 446.483,Z 101.178,A -85,B 0,C 180,E1 -8881.822,E2 -8881.822} C_VEL
LIN {X 0,Y 446.456,Z 101.184,A -85,B 0,C 180,E1 -8884.848,E2 -8884.848} C_VEL
LIN {X 0,Y 446.447,Z 101.187,A -85,B 0,C 180,E1 -8888.246,E2 -8888.246} C_VEL
LIN {X 0,Y 446.456,Z 101.181,A -85,B 0,C 180,E1 -8891.65,E2 -8891.65} C_VEL
LIN {X 0,Y 446.507,Z 101.18,A -85,B 0,C 180,E1 -8894.48,E2 -8894.48} C_VEL
LIN {X 0,Y 446.517,Z 101.18,A -85,B 0,C 180,E1 -8898.194,E2 -8898.194} C_VEL
LIN {X 0,Y 446.6,Z 101.166,A -85,B 0,C 180,E1 -8901.858,E2 -8901.858} C_VEL
LIN {X 0,Y 446.645,Z 101.16,A -85,B 0,C 180,E1 -8904.583,E2 -8904.583} C_VEL
LIN {X 0,Y 446.611,Z 101.161,A -85,B 0,C 180,E1 -8907.005,E2 -8907.005} C_VEL
LIN {X 0,Y 446.083,Z 101.233,A -85,B 0,C 180,E1 -8907.758,E2 -8907.758} C_VEL
LIN {X 0,Y 443.262,Z 101.579,A -85,B 0,C 180,E1 -8908.981,E2 -8908.981} C_VEL
LIN {X 0,Y 440.782,Z 101.894,A -85,B 0,C 180,E1 -8909.968,E2 -8909.968} C_VEL
LIN {X 0,Y 439.701,Z 102.023,A -85,B 0,C 180,E1 -8910.731,E2 -8910.731} C_VEL
LIN {X 0,Y 439.61,Z 102.033,A -85,B 0,C 180,E1 -8910.99,E2 -8910.99} C_VEL
LIN {X 0,Y 439.641,Z 102.03,A -85,B 0,C 180,E1 -8912.749,E2 -8912.749} C_VEL
LIN {X 0,Y 439.619,Z 102.034,A -85,B 0,C 180,E1 -8916.426,E2 -8916.426} C_VEL
LIN {X 0,Y 439.501,Z 102.048,A -85,B 0,C 180,E1 -8919.202,E2 -8919.202} C_VEL
LIN {X 0,Y 439.467,Z 102.051,A -85,B 0,C 180,E1 -8922.938,E2 -8922.938} C_VEL
LIN {X 0,Y 439.449,Z 102.055,A -85,B 0,C 180,E1 -8926.349,E2 -8926.349} C_VEL
LIN {X 0,Y 439.405,Z 102.066,A -85,B 0,C 180,E1 -8929.627,E2 -8929.627} C_VEL
LIN {X 0,Y 439.366,Z 102.064,A -85,B 0,C 180,E1 -8932.576,E2 -8932.576} C_VEL
LIN {X 0,Y 439.4,Z 102.067,A -85,B 0,C 180,E1 -8935.586,E2 -8935.586} C_VEL
LIN {X 0,Y 439.42,Z 102.057,A -85,B 0,C 180,E1 -8938.674,E2 -8938.674} C_VEL
LIN {X 0,Y 439.373,Z 102.065,A -85,B 0,C 180,E1 -8942.031,E2 -8942.031} C_VEL
LIN {X 0,Y 439.397,Z 102.066,A -85,B 0,C 180,E1 -8945.341,E2 -8945.341} C_VEL
LIN {X 0,Y 439.386,Z 102.062,A -85,B 0,C 180,E1 -8948.595,E2 -8948.595} C_VEL
LIN {X 0,Y 439.391,Z 102.067,A -85,B 0,C 180,E1 -8951.257,E2 -8951.257} C_VEL
LIN {X 0,Y 439.408,Z 102.06,A -85,B 0,C 180,E1 -8954.729,E2 -8954.729} C_VEL
LIN {X 0,Y 439.399,Z 102.061,A -85,B 0,C 180,E1 -8957.796,E2 -8957.796} C_VEL
LIN {X 0,Y 439.414,Z 102.058,A -85,B 0,C 180,E1 -8960.226,E2 -8960.226} C_VEL
LIN {X 0,Y 439.377,Z 102.067,A -85,B 0,C 180,E1 -8963.713,E2 -8963.713} C_VEL
LIN {X 0,Y 439.376,Z 102.069,A -85,B 0,C 180,E1 -8967.054,E2 -8967.054} C_VEL
LIN {X 0,Y 439.409,Z 102.066,A -85,B 0,C 180,E1 -8969.115,E2 -8969.115} C_VEL
LIN {X 0,Y 440.528,Z 105.079,A -85,B 0,C 180,E1 -8969.282,E2 -8969.282} C_VEL
LIN {X 0,Y 453.824,Z 131.5,A -85,B 0,C 180,E1 -8970.729,E2 -8970.729} C_VEL
LIN {X 0,Y 450.116,Z 276.443,A -85,B 0,C 180,E1 -8973.483,E2 -8973.483} C_VEL
LIN {X 0,Y 449.6,Z 297.357,A -85,B 0,C 180,E1 -8973.919,E2 -8973.919} C_VEL
LIN {X 0,Y 449.05,Z 313.423,A -85,B 0,C 180,E1 -8974.414,E2 -8974.414} C_VEL
LIN {X 0,Y 448.242,Z 330.087,A -85,B 0,C 180,E1 -8975.114,E2 -8975.114} C_VEL
LIN {X 0,Y 447.399,Z 344.621,A -85,B 0,C 180,E1 -8975.894,E2 -8975.894} C_VEL
LIN {X 0,Y 446.282,Z 360.539,A -85,B 0,C 180,E1 -8976.938,E2 -8976.938} C_VEL
LIN {X 0,Y 445.178,Z 375.142,A -85,B 0,C 180,E1 -8978.101,E2 -8978.101} C_VEL
LIN {X 0,Y 444.132,Z 387.836,A -85,B 0,C 180,E1 -8979.293,E2 -8979.293} C_VEL
LIN {X 0,Y 443.025,Z 401.188,A -85,B 0,C 180,E1 -8980.782,E2 -8980.782} C_VEL
LIN {X 0,Y 442.143,Z 411.875,A -85,B 0,C 180,E1 -8982.183,E2 -8982.183} C_VEL
LIN {X 0,Y 441.254,Z 422.629,A -85,B 0,C 180,E1 -8983.816,E2 -8983.816} C_VEL
LIN {X 0,Y 440.514,Z 431.832,A -85,B 0,C 180,E1 -8985.447,E2 -8985.447} C_VEL
LIN {X 0,Y 439.872,Z 440.286,A -85,B 0,C 180,E1 -8987.232,E2 -8987.232} C_VEL
LIN {X 0,Y 439.364,Z 447.091,A -85,B 0,C 180,E1 -8988.933,E2 -8988.933} C_VEL
LIN {X 0,Y 439.06,Z 453.27,A -85,B 0,C 180,E1 -8990.789,E2 -8990.789} C_VEL
LIN {X 0,Y 438.841,Z 458.141,A -85,B 0,C 180,E1 -8992.639,E2 -8992.639} C_VEL
LIN {X 0,Y 438.586,Z 461.949,A -85,B 0,C 180,E1 -8994.483,E2 -8994.483} C_VEL
LIN {X 0,Y 438.61,Z 464.665,A -85,B 0,C 180,E1 -8996.325,E2 -8996.325} C_VEL
LIN {X 0,Y 438.474,Z 466.361,A -85,B 0,C 180,E1 -8998.163,E2 -8998.163} C_VEL
LIN {X 0,Y 438.37,Z 467.104,A -85,B 0,C 180,E1 -9000,E2 -9000} C_VEL
LIN {X 0,Y 438.475,Z 466.774,A -85,B 0,C 180,E1 -9001.837,E2 -9001.837} C_VEL
LIN {X 0,Y 438.689,Z 465.521,A -85,B 0,C 180,E1 -9003.674,E2 -9003.674} C_VEL
LIN {X 0,Y 438.639,Z 463.183,A -85,B 0,C 180,E1 -9005.516,E2 -9005.516} C_VEL
LIN {X 0,Y 438.963,Z 459.842,A -85,B 0,C 180,E1 -9007.359,E2 -9007.359} C_VEL
LIN {X 0,Y 439.248,Z 455.37,A -85,B 0,C 180,E1 -9009.207,E2 -9009.207} C_VEL
LIN {X 0,Y 439.711,Z 449.692,A -85,B 0,C 180,E1 -9011.058,E2 -9011.058} C_VEL
LIN {X 0,Y 440.237,Z 442.763,A -85,B 0,C 180,E1 -9012.914,E2 -9012.914} C_VEL
LIN {X 0,Y 441.04,Z 434.339,A -85,B 0,C 180,E1 -9014.771,E2 -9014.771} C_VEL
LIN {X 0,Y 441.97,Z 424.174,A -85,B 0,C 180,E1 -9016.632,E2 -9016.632} C_VEL
LIN {X 0,Y 442.975,Z 413.582,A -85,B 0,C 180,E1 -9018.26,E2 -9018.26} C_VEL
LIN {X 0,Y 443.965,Z 402.99,A -85,B 0,C 180,E1 -9019.657,E2 -9019.657} C_VEL
LIN {X 0,Y 445.072,Z 390.872,A -85,B 0,C 180,E1 -9021.034,E2 -9021.034} C_VEL
LIN {X 0,Y 446.325,Z 377.339,A -85,B 0,C 180,E1 -9022.326,E2 -9022.326} C_VEL
LIN {X 0,Y 447.504,Z 362.855,A -85,B 0,C 180,E1 -9023.485,E2 -9023.485} C_VEL
LIN {X 0,Y 448.602,Z 347.824,A -85,B 0,C 180,E1 -9024.48,E2 -9024.48} C_VEL
LIN {X 0,Y 449.581,Z 331.847,A -85,B 0,C 180,E1 -9025.336,E2 -9025.336} C_VEL
LIN {X 0,Y 450.377,Z 316.073,A -85,B 0,C 180,E1 -9026.001,E2 -9026.001} C_VEL
LIN {X 0,Y 450.962,Z 300.652,A -85,B 0,C 180,E1 -9026.494,E2 -9026.494} C_VEL
LIN {X 0,Y 454.431,Z 214.313,A -85,B 0,C 180,E1 -9028.427,E2 -9028.427} C_VEL
LIN {X 0,Y 458.925,Z 135.532,A -85,B 0,C 180,E1 -9030.326,E2 -9030.326} C_VEL
LIN {X 0,Y 458.794,Z 134.297,A -85,B 0,C 180,E1 -9030.381,E2 -9030.381} C_VEL
LIN {X 0,Y 453.056,Z 123.569,A -85,B 0,C 180,E1 -9031.44,E2 -9031.44} C_VEL
LIN {X 0,Y 447.536,Z 114.83,A -85,B 0,C 180,E1 -9032.524,E2 -9032.524} C_VEL
LIN {X 0,Y 445.392,Z 111.489,A -85,B 0,C 180,E1 -9032.991,E2 -9032.991} C_VEL
LIN {X 0,Y 440.585,Z 105.165,A -85,B 0,C 180,E1 -9034.103,E2 -9034.103} C_VEL
LIN {X 0,Y 439.38,Z 102.069,A -85,B 0,C 180,E1 -9035.292,E2 -9035.292} C_VEL
LIN {X 0,Y 439.371,Z 102.069,A -85,B 0,C 180,E1 -9038.596,E2 -9038.596} C_VEL
LIN {X 0,Y 439.39,Z 102.066,A -85,B 0,C 180,E1 -9041.256,E2 -9041.256} C_VEL
LIN {X 0,Y 439.401,Z 102.066,A -85,B 0,C 180,E1 -9044.729,E2 -9044.729} C_VEL
LIN {X 0,Y 439.397,Z 102.066,A -85,B 0,C 180,E1 -9047.795,E2 -9047.795} C_VEL
LIN {X 0,Y 439.407,Z 102.097,A -85,B 0,C 180,E1 -9049.247,E2 -9049.247} C_VEL
LIN {X 0,Y 440.763,Z 105.394,A -85,B 0,C 180,E1 -9050.371,E2 -9050.371} C_VEL
LIN {X 0,Y 441.5,Z 107.083,A -85,B 0,C 180,E1 -9050.898,E2 -9050.898} C_VEL
LIN {X 0,Y 444.413,Z 113.835,A -85,B 0,C 180,E1 -9052.739,E2 -9052.739} C_VEL
LIN {X 0,Y 447.833,Z 122.607,A -85,B 0,C 180,E1 -9054.691,E2 -9054.691} C_VEL
LIN {X 0,Y 450.508,Z 130.813,A -85,B 0,C 180,E1 -9056.21,E2 -9056.21} C_VEL
LIN {X 0,Y 452.272,Z 137.603,A -85,B 0,C 180,E1 -9057.316,E2 -9057.316} C_VEL
LIN {X 0,Y 452.22,Z 140.063,A -85,B 0,C 180,E1 -9057.612,E2 -9057.612} C_VEL
LIN {X 0,Y 454.78,Z 157.465,A -85,B 0,C 180,E1 -9058.511,E2 -9058.511} C_VEL
LIN {X 0,Y 457.005,Z 179.056,A -85,B 0,C 180,E1 -9059.428,E2 -9059.428} C_VEL
LIN {X 0,Y 457.319,Z 185.353,A -85,B 0,C 180,E1 -9059.652,E2 -9059.652} C_VEL
LIN {X 0,Y 453.137,Z 268.353,A -85,B 0,C 180,E1 -9061.578,E2 -9061.578} C_VEL
LIN {X 0,Y 449.92,Z 356.391,A -85,B 0,C 180,E1 -9063.502,E2 -9063.502} C_VEL
LIN {X 0,Y 448.795,Z 374.274,A -85,B 0,C 180,E1 -9064.055,E2 -9064.055} C_VEL
LIN {X 0,Y 447.652,Z 391.676,A -85,B 0,C 180,E1 -9064.795,E2 -9064.795} C_VEL
LIN {X 0,Y 446.328,Z 408.622,A -85,B 0,C 180,E1 -9065.708,E2 -9065.708} C_VEL
LIN {X 0,Y 444.877,Z 425.785,A -85,B 0,C 180,E1 -9066.86,E2 -9066.86} C_VEL
LIN {X 0,Y 443.575,Z 441.417,A -85,B 0,C 180,E1 -9068.14,E2 -9068.14} C_VEL
LIN {X 0,Y 442.374,Z 456.393,A -85,B 0,C 180,E1 -9069.608,E2 -9069.608} C_VEL
LIN {X 0,Y 441.423,Z 468.04,A -85,B 0,C 180,E1 -9070.95,E2 -9070.95} C_VEL
LIN {X 0,Y 440.501,Z 480.342,A -85,B 0,C 180,E1 -9072.593,E2 -9072.593} C_VEL
LIN {X 0,Y 439.808,Z 490.89,A -85,B 0,C 180,E1 -9074.237,E2 -9074.237} C_VEL
LIN {X 0,Y 439.219,Z 501.071,A -85,B 0,C 180,E1 -9076.112,E2 -9076.112} C_VEL
LIN {X 0,Y 438.826,Z 509.524,A -85,B 0,C 180,E1 -9077.982,E2 -9077.982} C_VEL
LIN {X 0,Y 438.551,Z 516.534,A -85,B 0,C 180,E1 -9079.846,E2 -9079.846} C_VEL
LIN {X 0,Y 438.505,Z 522.281,A -85,B 0,C 180,E1 -9081.706,E2 -9081.706} C_VEL
LIN {X 0,Y 438.542,Z 526.714,A -85,B 0,C 180,E1 -9083.558,E2 -9083.558} C_VEL
LIN {X 0,Y 438.379,Z 530.03,A -85,B 0,C 180,E1 -9085.402,E2 -9085.402} C_VEL
LIN {X 0,Y 438.485,Z 532.244,A -85,B 0,C 180,E1 -9087.243,E2 -9087.243} C_VEL
LIN {X 0,Y 438.376,Z 533.361,A -85,B 0,C 180,E1 -9089.081,E2 -9089.081} C_VEL
LIN {X 0,Y 438.374,Z 533.451,A -85,B 0,C 180,E1 -9090.918,E2 -9090.918} C_VEL
LIN {X 0,Y 438.468,Z 532.443,A -85,B 0,C 180,E1 -9092.756,E2 -9092.756} C_VEL
LIN {X 0,Y 438.36,Z 530.413,A -85,B 0,C 180,E1 -9094.597,E2 -9094.597} C_VEL
LIN {X 0,Y 438.502,Z 527.222,A -85,B 0,C 180,E1 -9096.441,E2 -9096.441} C_VEL
LIN {X 0,Y 438.494,Z 522.941,A -85,B 0,C 180,E1 -9098.293,E2 -9098.293} C_VEL
LIN {X 0,Y 438.549,Z 517.396,A -85,B 0,C 180,E1 -9100.153,E2 -9100.153} C_VEL
LIN {X 0,Y 438.857,Z 510.547,A -85,B 0,C 180,E1 -9102.015,E2 -9102.015} C_VEL
LIN {X 0,Y 439.263,Z 502.264,A -85,B 0,C 180,E1 -9103.885,E2 -9103.885} C_VEL
LIN {X 0,Y 439.864,Z 492.322,A -85,B 0,C 180,E1 -9105.76,E2 -9105.76} C_VEL
LIN {X 0,Y 440.62,Z 482,A -85,B 0,C 180,E1 -9107.401,E2 -9107.401} C_VEL
LIN {X 0,Y 441.56,Z 469.854,A -85,B 0,C 180,E1 -9109.043,E2 -9109.043} C_VEL
LIN {X 0,Y 442.633,Z 457.332,A -85,B 0,C 180,E1 -9110.482,E2 -9110.482} C_VEL
LIN {X 0,Y 443.772,Z 443.349,A -85,B 0,C 180,E1 -9111.849,E2 -9111.849} C_VEL
LIN {X 0,Y 444.944,Z 429.204,A -85,B 0,C 180,E1 -9113.012,E2 -9113.012} C_VEL
LIN {X 0,Y 446.183,Z 413.709,A -85,B 0,C 180,E1 -9114.067,E2 -9114.067} C_VEL
LIN {X 0,Y 447.353,Z 397.173,A -85,B 0,C 180,E1 -9114.974,E2 -9114.974} C_VEL
LIN {X 0,Y 448.335,Z 380.334,A -85,B 0,C 180,E1 -9115.691,E2 -9115.691} C_VEL
LIN {X 0,Y 449.174,Z 364.033,A -85,B 0,C 180,E1 -9116.2,E2 -9116.2} C_VEL
LIN {X 0,Y 449.888,Z 342.302,A -85,B 0,C 180,E1 -9116.655,E2 -9116.655} C_VEL
LIN {X 0,Y 453.941,Z 183.349,A -85,B 0,C 180,E1 -9119.681,E2 -9119.681} C_VEL
LIN {X 0,Y 449.433,Z 151.181,A -85,B 0,C 180,E1 -9120.677,E2 -9120.677} C_VEL
LIN {X 0,Y 450.382,Z 137.423,A -85,B 0,C 180,E1 -9122.042,E2 -9122.042} C_VEL
LIN {X 0,Y 449.706,Z 133.986,A -85,B 0,C 180,E1 -9122.445,E2 -9122.445} C_VEL
LIN {X 0,Y 443.633,Z 114.909,A -85,B 0,C 180,E1 -9124.9,E2 -9124.9} C_VEL
LIN {X 0,Y 439.357,Z 102.072,A -85,B 0,C 180,E1 -9126.644,E2 -9126.644} C_VEL
LIN {X 0,Y 439.397,Z 102.065,A -85,B 0,C 180,E1 -9129.849,E2 -9129.849} C_VEL
LIN {X 0,Y 439.399,Z 102.067,A -85,B 0,C 180,E1 -9132.63,E2 -9132.63} C_VEL
LIN {X 0,Y 439.398,Z 102.063,A -85,B 0,C 180,E1 -9135.271,E2 -9135.271} C_VEL
LIN {X 0,Y 439.384,Z 102.065,A -85,B 0,C 180,E1 -9138.743,E2 -9138.743} C_VEL
LIN {X 0,Y 439.381,Z 102.063,A -85,B 0,C 180,E1 -9141.606,E2 -9141.606} C_VEL
LIN {X 0,Y 439.396,Z 102.061,A -85,B 0,C 180,E1 -9144.844,E2 -9144.844} C_VEL
LIN {X 0,Y 439.381,Z 102.069,A -85,B 0,C 180,E1 -9148.14,E2 -9148.14} C_VEL
LIN {X 0,Y 439.42,Z 102.057,A -85,B 0,C 180,E1 -9151.327,E2 -9151.327} C_VEL
LIN {X 0,Y 439.401,Z 102.063,A -85,B 0,C 180,E1 -9154.415,E2 -9154.415} C_VEL
LIN {X 0,Y 439.361,Z 102.066,A -85,B 0,C 180,E1 -9157.425,E2 -9157.425} C_VEL
LIN {X 0,Y 439.437,Z 102.056,A -85,B 0,C 180,E1 -9160.663,E2 -9160.663} C_VEL
LIN {X 0,Y 439.471,Z 102.054,A -85,B 0,C 180,E1 -9164.225,E2 -9164.225} C_VEL
LIN {X 0,Y 439.503,Z 102.052,A -85,B 0,C 180,E1 -9168.002,E2 -9168.002} C_VEL
LIN {X 0,Y 439.543,Z 102.049,A -85,B 0,C 180,E1 -9171.726,E2 -9171.726} C_VEL
LIN {X 0,Y 439.616,Z 102.033,A -85,B 0,C 180,E1 -9174.496,E2 -9174.496} C_VEL
LIN {X 0,Y 439.632,Z 102.033,A -85,B 0,C 180,E1 -9178.168,E2 -9178.168} C_VEL
LIN {X 0,Y 439.759,Z 102.018,A -85,B 0,C 180,E1 -9180,E2 -9180} C_VEL
LIN {X 0,Y 439.652,Z 102.028,A -85,B 0,C 180,E1 -9182.749,E2 -9182.749} C_VEL
LIN {X 0,Y 439.614,Z 102.033,A -85,B 0,C 180,E1 -9186.425,E2 -9186.425} C_VEL
LIN {X 0,Y 439.495,Z 102.052,A -85,B 0,C 180,E1 -9189.202,E2 -9189.202} C_VEL
LIN {X 0,Y 439.461,Z 102.054,A -85,B 0,C 180,E1 -9192.938,E2 -9192.938} C_VEL
LIN {X 0,Y 439.443,Z 102.054,A -85,B 0,C 180,E1 -9196.349,E2 -9196.349} C_VEL
LIN {X 0,Y 439.398,Z 102.063,A -85,B 0,C 180,E1 -9199.626,E2 -9199.626} C_VEL
LIN {X 0,Y 439.361,Z 102.065,A -85,B 0,C 180,E1 -9202.576,E2 -9202.576} C_VEL
LIN {X 0,Y 439.401,Z 102.062,A -85,B 0,C 180,E1 -9205.585,E2 -9205.585} C_VEL
LIN {X 0,Y 439.413,Z 102.06,A -85,B 0,C 180,E1 -9208.674,E2 -9208.674} C_VEL
LIN {X 0,Y 439.367,Z 102.064,A -85,B 0,C 180,E1 -9212.031,E2 -9212.031} C_VEL
LIN {X 0,Y 439.392,Z 102.064,A -85,B 0,C 180,E1 -9215.341,E2 -9215.341} C_VEL
LIN {X 0,Y 439.385,Z 102.065,A -85,B 0,C 180,E1 -9218.595,E2 -9218.595} C_VEL
LIN {X 0,Y 439.386,Z 102.065,A -85,B 0,C 180,E1 -9221.257,E2 -9221.257} C_VEL
LIN {X 0,Y 439.403,Z 102.065,A -85,B 0,C 180,E1 -9224.729,E2 -9224.729} C_VEL
LIN {X 0,Y 439.395,Z 102.06,A -85,B 0,C 180,E1 -9227.797,E2 -9227.797} C_VEL
LIN {X 0,Y 439.442,Z 102.056,A -85,B 0,C 180,E1 -9230.23,E2 -9230.23} C_VEL
LIN {X 0,Y 439.371,Z 102.063,A -85,B 0,C 180,E1 -9233.713,E2 -9233.713} C_VEL
LIN {X 0,Y 439.37,Z 102.066,A -85,B 0,C 180,E1 -9237.055,E2 -9237.055} C_VEL
LIN {X 0,Y 439.381,Z 102.066,A -85,B 0,C 180,E1 -9240.275,E2 -9240.275} C_VEL
LIN {X 0,Y 439.428,Z 102.056,A -85,B 0,C 180,E1 -9243.397,E2 -9243.397} C_VEL
LIN {X 0,Y 439.386,Z 102.069,A -85,B 0,C 180,E1 -9246.43,E2 -9246.43} C_VEL
LIN {X 0,Y 439.387,Z 102.061,A -85,B 0,C 180,E1 -9249.398,E2 -9249.398} C_VEL
LIN {X 0,Y 439.431,Z 102.063,A -85,B 0,C 180,E1 -9252.31,E2 -9252.31} C_VEL
LIN {X 0,Y 439.447,Z 102.054,A -85,B 0,C 180,E1 -9255.175,E2 -9255.175} C_VEL
LIN {X 0,Y 439.483,Z 102.053,A -85,B 0,C 180,E1 -9258.002,E2 -9258.002} C_VEL
LIN {X 0,Y 439.548,Z 102.043,A -85,B 0,C 180,E1 -9261.727,E2 -9261.727} C_VEL
LIN {X 0,Y 439.621,Z 102.035,A -85,B 0,C 180,E1 -9264.496,E2 -9264.496} C_VEL
LIN {X 0,Y 439.635,Z 102.037,A -85,B 0,C 180,E1 -9268.168,E2 -9268.168} C_VEL
LIN {X 0,Y 439.763,Z 102.021,A -85,B 0,C 180,E1 -9270.001,E2 -9270.001} C_VEL
LIN {X 0,Y 439.61,Z 102.033,A -85,B 0,C 180,E1 -9270.99,E2 -9270.99} C_VEL
LIN {X 0,Y 438.901,Z 102.128,A -85,B 0,C 180,E1 -9271.754,E2 -9271.754} C_VEL
LIN {X 0,Y 435.926,Z 102.492,A -85,B 0,C 180,E1 -9272.993,E2 -9272.993} C_VEL
LIN {X 0,Y 433.474,Z 102.806,A -85,B 0,C 180,E1 -9273.994,E2 -9273.994} C_VEL
LIN {X 0,Y 432.501,Z 102.92,A -85,B 0,C 180,E1 -9274.769,E2 -9274.769} C_VEL
LIN {X 0,Y 432.464,Z 102.924,A -85,B 0,C 180,E1 -9275.031,E2 -9275.031} C_VEL
LIN {X 0,Y 432.587,Z 102.913,A -85,B 0,C 180,E1 -9277.68,E2 -9277.68} C_VEL
LIN {X 0,Y 432.394,Z 102.934,A -85,B 0,C 180,E1 -9281.248,E2 -9281.248} C_VEL
LIN {X 0,Y 432.375,Z 102.939,A -85,B 0,C 180,E1 -9284.112,E2 -9284.112} C_VEL
LIN {X 0,Y 432.399,Z 102.932,A -85,B 0,C 180,E1 -9287.012,E2 -9287.012} C_VEL
LIN {X 0,Y 432.341,Z 102.943,A -85,B 0,C 180,E1 -9289.961,E2 -9289.961} C_VEL
LIN {X 0,Y 432.32,Z 102.942,A -85,B 0,C 180,E1 -9292.965,E2 -9292.965} C_VEL
LIN {X 0,Y 432.363,Z 102.939,A -85,B 0,C 180,E1 -9296.033,E2 -9296.033} C_VEL
LIN {X 0,Y 432.346,Z 102.942,A -85,B 0,C 180,E1 -9299.188,E2 -9299.188} C_VEL
LIN {X 0,Y 432.325,Z 102.941,A -85,B 0,C 180,E1 -9302.443,E2 -9302.443} C_VEL
LIN {X 0,Y 432.346,Z 102.943,A -85,B 0,C 180,E1 -9305.632,E2 -9305.632} C_VEL
LIN {X 0,Y 432.353,Z 102.945,A -85,B 0,C 180,E1 -9309.343,E2 -9309.343} C_VEL
LIN {X 0,Y 432.337,Z 102.942,A -85,B 0,C 180,E1 -9311.797,E2 -9311.797} C_VEL
LIN {X 0,Y 432.343,Z 102.939,A -85,B 0,C 180,E1 -9314.347,E2 -9314.347} C_VEL
LIN {X 0,Y 432.323,Z 102.946,A -85,B 0,C 180,E1 -9317.016,E2 -9317.016} C_VEL
LIN {X 0,Y 432.336,Z 102.941,A -85,B 0,C 180,E1 -9319.821,E2 -9319.821} C_VEL
LIN {X 0,Y 432.31,Z 102.949,A -85,B 0,C 180,E1 -9323.022,E2 -9323.022} C_VEL
LIN {X 0,Y 432.363,Z 102.938,A -85,B 0,C 180,E1 -9325.997,E2 -9325.997} C_VEL
LIN {X 0,Y 432.354,Z 102.942,A -85,B 0,C 180,E1 -9328.657,E2 -9328.657} C_VEL
LIN {X 0,Y 433.369,Z 105.82,A -85,B 0,C 180,E1 -9328.803,E2 -9328.803} C_VEL
LIN {X 0,Y 447.462,Z 133.801,A -85,B 0,C 180,E1 -9330.372,E2 -9330.372} C_VEL
LIN {X 0,Y 443.372,Z 283.361,A -85,B 0,C 180,E1 -9333.27,E2 -9333.27} C_VEL
LIN {X 0,Y 442.873,Z 301.081,A -85,B 0,C 180,E1 -9333.683,E2 -9333.683} C_VEL
LIN {X 0,Y 442.151,Z 318.324,A -85,B 0,C 180,E1 -9334.27,E2 -9334.27} C_VEL
LIN {X 0,Y 441.275,Z 335.509,A -85,B 0,C 180,E1 -9335.062,E2 -9335.062} C_VEL
LIN {X 0,Y 440.292,Z 351.21,A -85,B 0,C 180,E1 -9335.981,E2 -9335.981} C_VEL
LIN {X 0,Y 439.197,Z 366.092,A -85,B 0,C 180,E1 -9337.043,E2 -9337.043} C_VEL
LIN {X 0,Y 438.107,Z 379.901,A -85,B 0,C 180,E1 -9338.225,E2 -9338.225} C_VEL
LIN {X 0,Y 436.956,Z 392.724,A -85,B 0,C 180,E1 -9339.523,E2 -9339.523} C_VEL
LIN {X 0,Y 435.886,Z 404.73,A -85,B 0,C 180,E1 -9340.943,E2 -9340.943} C_VEL
LIN {X 0,Y 434.887,Z 416.657,A -85,B 0,C 180,E1 -9342.603,E2 -9342.603} C_VEL
LIN {X 0,Y 434.013,Z 426.826,A -85,B 0,C 180,E1 -9344.262,E2 -9344.262} C_VEL
LIN {X 0,Y 433.199,Z 436.564,A -85,B 0,C 180,E1 -9346.155,E2 -9346.155} C_VEL
LIN {X 0,Y 432.68,Z 443.729,A -85,B 0,C 180,E1 -9347.81,E2 -9347.81} C_VEL
LIN {X 0,Y 432.189,Z 450.636,A -85,B 0,C 180,E1 -9349.696,E2 -9349.696} C_VEL
LIN {X 0,Y 431.893,Z 456.195,A -85,B 0,C 180,E1 -9351.579,E2 -9351.579} C_VEL
LIN {X 0,Y 431.712,Z 460.578,A -85,B 0,C 180,E1 -9353.457,E2 -9353.457} C_VEL
LIN {X 0,Y 431.521,Z 463.925,A -85,B 0,C 180,E1 -9355.329,E2 -9355.329} C_VEL
LIN {X 0,Y 431.52,Z 466.125,A -85,B 0,C 180,E1 -9357.199,E2 -9357.199} C_VEL
LIN {X 0,Y 431.332,Z 467.414,A -85,B 0,C 180,E1 -9359.066,E2 -9359.066} C_VEL
LIN {X 0,Y 431.334,Z 467.624,A -85,B 0,C 180,E1 -9360.933,E2 -9360.933} C_VEL
LIN {X 0,Y 431.584,Z 466.864,A -85,B 0,C 180,E1 -9362.8,E2 -9362.8} C_VEL
LIN {X 0,Y 431.652,Z 465.094,A -85,B 0,C 180,E1 -9364.669,E2 -9364.669} C_VEL
LIN {X 0,Y 431.866,Z 461.567,A -85,B 0,C 180,E1 -9366.93,E2 -9366.93} C_VEL
LIN {X 0,Y 432.164,Z 457.255,A -85,B 0,C 180,E1 -9368.887,E2 -9368.887} C_VEL
LIN {X 0,Y 432.628,Z 451.967,A -85,B 0,C 180,E1 -9370.767,E2 -9370.767} C_VEL
LIN {X 0,Y 433.167,Z 445.336,A -85,B 0,C 180,E1 -9372.652,E2 -9372.652} C_VEL
LIN {X 0,Y 433.94,Z 437.289,A -85,B 0,C 180,E1 -9374.539,E2 -9374.539} C_VEL
LIN {X 0,Y 434.917,Z 427.624,A -85,B 0,C 180,E1 -9376.427,E2 -9376.427} C_VEL
LIN {X 0,Y 435.915,Z 417.759,A -85,B 0,C 180,E1 -9378.056,E2 -9378.056} C_VEL
LIN {X 0,Y 437.153,Z 405.766,A -85,B 0,C 180,E1 -9379.731,E2 -9379.731} C_VEL
LIN {X 0,Y 438.397,Z 393.03,A -85,B 0,C 180,E1 -9381.229,E2 -9381.229} C_VEL
LIN {X 0,Y 439.725,Z 379.581,A -85,B 0,C 180,E1 -9382.556,E2 -9382.556} C_VEL
LIN {X 0,Y 440.966,Z 365.484,A -85,B 0,C 180,E1 -9383.73,E2 -9383.73} C_VEL
LIN {X 0,Y 441.988,Z 352.482,A -85,B 0,C 180,E1 -9384.646,E2 -9384.646} C_VEL
LIN {X 0,Y 443.135,Z 336.971,A -85,B 0,C 180,E1 -9385.543,E2 -9385.543} C_VEL
LIN {X 0,Y 444.058,Z 319.665,A -85,B 0,C 180,E1 -9386.336,E2 -9386.336} C_VEL
LIN {X 0,Y 444.837,Z 302.282,A -85,B 0,C 180,E1 -9386.919,E2 -9386.919} C_VEL
LIN {X 0,Y 448.529,Z 217.883,A -85,B 0,C 180,E1 -9388.884,E2 -9388.884} C_VEL
LIN {X 0,Y 453.556,Z 138.596,A -85,B 0,C 180,E1 -9390.85,E2 -9390.85} C_VEL
LIN {X 0,Y 453.507,Z 137.333,A -85,B 0,C 180,E1 -9390.899,E2 -9390.899} C_VEL
LIN {X 0,Y 448.542,Z 128.041,A -85,B 0,C 180,E1 -9391.865,E2 -9391.865} C_VEL
LIN {X 0,Y 443.532,Z 119.869,A -85,B 0,C 180,E1 -9392.925,E2 -9392.925} C_VEL
LIN {X 0,Y 441.632,Z 116.921,A -85,B 0,C 180,E1 -9393.355,E2 -9393.355} C_VEL
LIN {X 0,Y 437.303,Z 111.123,A -85,B 0,C 180,E1 -9394.39,E2 -9394.39} C_VEL
LIN {X 0,Y 434.651,Z 107.962,A -85,B 0,C 180,E1 -9395.079,E2 -9395.079} C_VEL
LIN {X 0,Y 434.174,Z 107.118,A -85,B 0,C 180,E1 -9395.258,E2 -9395.258} C_VEL
LIN {X 0,Y 432.45,Z 103.763,A -85,B 0,C 180,E1 -9396.963,E2 -9396.963} C_VEL
LIN {X 0,Y 432.312,Z 102.95,A -85,B 0,C 180,E1 -9397.371,E2 -9397.371} C_VEL
LIN {X 0,Y 432.326,Z 102.946,A -85,B 0,C 180,E1 -9400.56,E2 -9400.56} C_VEL
LIN {X 0,Y 432.319,Z 102.947,A -85,B 0,C 180,E1 -9403.06,E2 -9403.06} C_VEL
LIN {X 0,Y 432.335,Z 102.947,A -85,B 0,C 180,E1 -9405.664,E2 -9405.664} C_VEL
LIN {X 0,Y 432.332,Z 102.978,A -85,B 0,C 180,E1 -9407.185,E2 -9407.185} C_VEL
LIN {X 0,Y 433.131,Z 105.389,A -85,B 0,C 180,E1 -9408.297,E2 -9408.297} C_VEL
LIN {X 0,Y 434.555,Z 108.062,A -85,B 0,C 180,E1 -9409.475,E2 -9409.475} C_VEL
LIN {X 0,Y 436.182,Z 111.394,A -85,B 0,C 180,E1 -9410.66,E2 -9410.66} C_VEL
LIN {X 0,Y 439.272,Z 118.939,A -85,B 0,C 180,E1 -9412.764,E2 -9412.764} C_VEL
LIN {X 0,Y 442.447,Z 127.43,A -85,B 0,C 180,E1 -9414.673,E2 -9414.673} C_VEL
LIN {X 0,Y 444.867,Z 135.397,A -85,B 0,C 180,E1 -9416.159,E2 -9416.159} C_VEL
LIN {X 0,Y 445.904,Z 138.963,A -85,B 0,C 180,E1 -9416.734,E2 -9416.734} C_VEL
LIN {X 0,Y 447.221,Z 142.627,A -85,B 0,C 180,E1 -9417.054,E2 -9417.054} C_VEL
LIN {X 0,Y 449.533,Z 159.306,A -85,B 0,C 180,E1 -9417.95,E2 -9417.95} C_VEL
LIN {X 0,Y 451.455,Z 179.893,A -85,B 0,C 180,E1 -9418.865,E2 -9418.865} C_VEL
LIN {X 0,Y 451.742,Z 186.631,A -85,B 0,C 180,E1 -9419.109,E2 -9419.109} C_VEL
LIN {X 0,Y 447.379,Z 265.793,A -85,B 0,C 180,E1 -9421.018,E2 -9421.018} C_VEL
LIN {X 0,Y 444.434,Z 338.437,A -85,B 0,C 180,E1 -9422.647,E2 -9422.647} C_VEL
LIN {X 0,Y 443.528,Z 359.183,A -85,B 0,C 180,E1 -9423.153,E2 -9423.153} C_VEL
LIN {X 0,Y 442.254,Z 376.613,A -85,B 0,C 180,E1 -9423.738,E2 -9423.738} C_VEL
LIN {X 0,Y 440.944,Z 394.854,A -85,B 0,C 180,E1 -9424.573,E2 -9424.573} C_VEL
LIN {X 0,Y 439.543,Z 411.155,A -85,B 0,C 180,E1 -9425.512,E2 -9425.512} C_VEL
LIN {X 0,Y 438.119,Z 426.764,A -85,B 0,C 180,E1 -9426.607,E2 -9426.607} C_VEL
LIN {X 0,Y 436.923,Z 440.858,A -85,B 0,C 180,E1 -9427.789,E2 -9427.789} C_VEL
LIN {X 0,Y 435.652,Z 455.173,A -85,B 0,C 180,E1 -9429.212,E2 -9429.212} C_VEL
LIN {X 0,Y 434.564,Z 467.418,A -85,B 0,C 180,E1 -9430.637,E2 -9430.637} C_VEL
LIN {X 0,Y 433.577,Z 479.713,A -85,B 0,C 180,E1 -9432.306,E2 -9432.306} C_VEL
LIN {X 0,Y 432.795,Z 490.259,A -85,B 0,C 180,E1 -9433.974,E2 -9433.974} C_VEL
LIN {X 0,Y 432.199,Z 500.462,A -85,B 0,C 180,E1 -9435.882,E2 -9435.882} C_VEL
LIN {X 0,Y 431.772,Z 508.927,A -85,B 0,C 180,E1 -9437.783,E2 -9437.783} C_VEL
LIN {X 0,Y 431.494,Z 515.949,A -85,B 0,C 180,E1 -9439.678,E2 -9439.678} C_VEL
LIN {X 0,Y 431.405,Z 521.705,A -85,B 0,C 180,E1 -9441.568,E2 -9441.568} C_VEL
LIN {X 0,Y 431.458,Z 526.312,A -85,B 0,C 180,E1 -9443.525,E2 -9443.525} C_VEL
LIN {X 0,Y 431.304,Z 529.478,A -85,B 0,C 180,E1 -9445.326,E2 -9445.326} C_VEL
LIN {X 0,Y 431.409,Z 531.7,A -85,B 0,C 180,E1 -9447.198,E2 -9447.198} C_VEL
LIN {X 0,Y 431.317,Z 532.814,A -85,B 0,C 180,E1 -9449.066,E2 -9449.066} C_VEL
LIN {X 0,Y 431.315,Z 532.903,A -85,B 0,C 180,E1 -9450.933,E2 -9450.933} C_VEL
LIN {X 0,Y 431.394,Z 531.871,A -85,B 0,C 180,E1 -9452.801,E2 -9452.801} C_VEL
LIN {X 0,Y 431.285,Z 529.823,A -85,B 0,C 180,E1 -9454.673,E2 -9454.673} C_VEL
LIN {X 0,Y 431.432,Z 526.599,A -85,B 0,C 180,E1 -9456.547,E2 -9456.547} C_VEL
LIN {X 0,Y 431.397,Z 522.27,A -85,B 0,C 180,E1 -9458.431,E2 -9458.431} C_VEL
LIN {X 0,Y 431.492,Z 516.697,A -85,B 0,C 180,E1 -9460.32,E2 -9460.32} C_VEL
LIN {X 0,Y 431.807,Z 509.787,A -85,B 0,C 180,E1 -9462.215,E2 -9462.215} C_VEL
LIN {X 0,Y 432.232,Z 501.429,A -85,B 0,C 180,E1 -9464.116,E2 -9464.116} C_VEL
LIN {X 0,Y 432.796,Z 492.774,A -85,B 0,C 180,E1 -9465.782,E2 -9465.782} C_VEL
LIN {X 0,Y 433.542,Z 482.552,A -85,B 0,C 180,E1 -9467.451,E2 -9467.451} C_VEL
LIN {X 0,Y 434.522,Z 470.587,A -85,B 0,C 180,E1 -9469.118,E2 -9469.118} C_VEL
LIN {X 0,Y 435.669,Z 457.436,A -85,B 0,C 180,E1 -9470.671,E2 -9470.671} C_VEL
LIN {X 0,Y 436.905,Z 443.234,A -85,B 0,C 180,E1 -9472.086,E2 -9472.086} C_VEL
LIN {X 0,Y 438.115,Z 429.169,A -85,B 0,C 180,E1 -9473.266,E2 -9473.266} C_VEL
LIN {X 0,Y 439.33,Z 414.453,A -85,B 0,C 180,E1 -9474.291,E2 -9474.291} C_VEL
LIN {X 0,Y 440.531,Z 398.47,A -85,B 0,C 180,E1 -9475.198,E2 -9475.198} C_VEL
LIN {X 0,Y 441.564,Z 382.248,A -85,B 0,C 180,E1 -9475.924,E2 -9475.924} C_VEL
LIN {X 0,Y 442.468,Z 365.989,A -85,B 0,C 180,E1 -9476.47,E2 -9476.47} C_VEL
LIN {X 0,Y 443.142,Z 348.627,A -85,B 0,C 180,E1 -9476.871,E2 -9476.871} C_VEL
LIN {X 0,Y 447.564,Z 184.806,A -85,B 0,C 180,E1 -9480.055,E2 -9480.055} C_VEL
LIN {X 0,Y 442.904,Z 150.863,A -85,B 0,C 180,E1 -9481.112,E2 -9481.112} C_VEL
LIN {X 0,Y 443.761,Z 138.983,A -85,B 0,C 180,E1 -9482.31,E2 -9482.31} C_VEL
LIN {X 0,Y 440.152,Z 126.698,A -85,B 0,C 180,E1 -9483.871,E2 -9483.871} C_VEL
LIN {X 0,Y 434.086,Z 108.594,A -85,B 0,C 180,E1 -9486.31,E2 -9486.31} C_VEL
LIN {X 0,Y 432.319,Z 102.947,A -85,B 0,C 180,E1 -9487.113,E2 -9487.113} C_VEL
LIN {X 0,Y 432.33,Z 102.947,A -85,B 0,C 180,E1 -9490.179,E2 -9490.179} C_VEL
LIN {X 0,Y 432.361,Z 102.94,A -85,B 0,C 180,E1 -9493.055,E2 -9493.055} C_VEL
LIN {X 0,Y 432.328,Z 102.944,A -85,B 0,C 180,E1 -9495.664,E2 -9495.664} C_VEL
LIN {X 0,Y 432.329,Z 102.948,A -85,B 0,C 180,E1 -9498.398,E2 -9498.398} C_VEL
LIN {X 0,Y 432.343,Z 102.941,A -85,B 0,C 180,E1 -9501.851,E2 -9501.851} C_VEL
LIN {X 0,Y 432.336,Z 102.94,A -85,B 0,C 180,E1 -9505.323,E2 -9505.323} C_VEL
LIN {X 0,Y 432.324,Z 102.943,A -85,B 0,C 180,E1 -9508.654,E2 -9508.654} C_VEL
LIN {X 0,Y 432.379,Z 102.939,A -85,B 0,C 180,E1 -9511.877,E2 -9511.877} C_VEL
LIN {X 0,Y 432.347,Z 102.938,A -85,B 0,C 180,E1 -9514.999,E2 -9514.999} C_VEL
LIN {X 0,Y 432.354,Z 102.945,A -85,B 0,C 180,E1 -9518.046,E2 -9518.046} C_VEL
LIN {X 0,Y 432.382,Z 102.934,A -85,B 0,C 180,E1 -9521.03,E2 -9521.03} C_VEL
LIN {X 0,Y 432.438,Z 102.934,A -85,B 0,C 180,E1 -9523.962,E2 -9523.962} C_VEL
LIN {X 0,Y 432.476,Z 102.929,A -85,B 0,C 180,E1 -9527.804,E2 -9527.804} C_VEL
LIN {X 0,Y 432.487,Z 102.926,A -85,B 0,C 180,E1 -9531.59,E2 -9531.59} C_VEL
LIN {X 0,Y 432.593,Z 102.908,A -85,B 0,C 180,E1 -9534.406,E2 -9534.406} C_VEL
LIN {X 0,Y 432.601,Z 102.909,A -85,B 0,C 180,E1 -9538.138,E2 -9538.138} C_VEL
LIN {X 0,Y 432.729,Z 102.894,A -85,B 0,C 180,E1 -9540,E2 -9540} C_VEL
LIN {X 0,Y 432.601,Z 102.907,A -85,B 0,C 180,E1 -9542.794,E2 -9542.794} C_VEL
LIN {X 0,Y 432.568,Z 102.911,A -85,B 0,C 180,E1 -9546.53,E2 -9546.53} C_VEL
LIN {X 0,Y 432.438,Z 102.933,A -85,B 0,C 180,E1 -9549.353,E2 -9549.353} C_VEL
LIN {X 0,Y 432.426,Z 102.93,A -85,B 0,C 180,E1 -9552.804,E2 -9552.804} C_VEL
LIN {X 0,Y 432.408,Z 102.931,A -85,B 0,C 180,E1 -9556.479,E2 -9556.479} C_VEL
LIN {X 0,Y 432.335,Z 102.941,A -85,B 0,C 180,E1 -9559.961,E2 -9559.961} C_VEL
LIN {X 0,Y 432.316,Z 102.946,A -85,B 0,C 180,E1 -9562.964,E2 -9562.964} C_VEL
LIN {X 0,Y 432.36,Z 102.937,A -85,B 0,C 180,E1 -9566.033,E2 -9566.033} C_VEL
LIN {X 0,Y 432.339,Z 102.946,A -85,B 0,C 180,E1 -9569.188,E2 -9569.188} C_VEL
LIN {X 0,Y 432.319,Z 102.943,A -85,B 0,C 180,E1 -9572.443,E2 -9572.443} C_VEL
LIN {X 0,Y 432.342,Z 102.94,A -85,B 0,C 180,E1 -9575.633,E2 -9575.633} C_VEL
LIN {X 0,Y 432.347,Z 102.943,A -85,B 0,C 180,E1 -9578.717,E2 -9578.717} C_VEL
LIN {X 0,Y 432.331,Z 102.94,A -85,B 0,C 180,E1 -9581.797,E2 -9581.797} C_VEL
LIN {X 0,Y 432.338,Z 102.941,A -85,B 0,C 180,E1 -9584.347,E2 -9584.347} C_VEL
LIN {X 0,Y 432.322,Z 102.946,A -85,B 0,C 180,E1 -9587.016,E2 -9587.016} C_VEL
LIN {X 0,Y 432.349,Z 102.938,A -85,B 0,C 180,E1 -9589.818,E2 -9589.818} C_VEL
LIN {X 0,Y 432.304,Z 102.947,A -85,B 0,C 180,E1 -9593.023,E2 -9593.023} C_VEL
LIN {X 0,Y 432.356,Z 102.938,A -85,B 0,C 180,E1 -9595.997,E2 -9595.997} C_VEL
LIN {X 0,Y 432.345,Z 102.938,A -85,B 0,C 180,E1 -9599.49,E2 -9599.49} C_VEL
LIN {X 0,Y 432.39,Z 102.936,A -85,B 0,C 180,E1 -9602.929,E2 -9602.929} C_VEL
LIN {X 0,Y 432.37,Z 102.938,A -85,B 0,C 180,E1 -9606.024,E2 -9606.024} C_VEL
LIN {X 0,Y 432.349,Z 102.939,A -85,B 0,C 180,E1 -9609.047,E2 -9609.047} C_VEL
LIN {X 0,Y 432.377,Z 102.938,A -85,B 0,C 180,E1 -9612.012,E2 -9612.012} C_VEL
LIN {X 0,Y 432.395,Z 102.933,A -85,B 0,C 180,E1 -9614.927,E2 -9614.927} C_VEL
LIN {X 0,Y 432.459,Z 102.926,A -85,B 0,C 180,E1 -9617.804,E2 -9617.804} C_VEL
LIN {X 0,Y 432.492,Z 102.921,A -85,B 0,C 180,E1 -9621.591,E2 -9621.591} C_VEL
LIN {X 0,Y 432.597,Z 102.911,A -85,B 0,C 180,E1 -9624.407,E2 -9624.407} C_VEL
LIN {X 0,Y 432.604,Z 102.913,A -85,B 0,C 180,E1 -9628.139,E2 -9628.139} C_VEL
LIN {X 0,Y 432.733,Z 102.897,A -85,B 0,C 180,E1 -9630.001,E2 -9630.001} C_VEL
LIN {X 0,Y 432.593,Z 102.908,A -85,B 0,C 180,E1 -9632.794,E2 -9632.794} C_VEL
LIN {X 0,Y 432.464,Z 102.924,A -85,B 0,C 180,E1 -9635.031,E2 -9635.031} C_VEL
LIN {X 0,Y 431.906,Z 102.999,A -85,B 0,C 180,E1 -9635.809,E2 -9635.809} C_VEL
LIN {X 0,Y 429.061,Z 103.348,A -85,B 0,C 180,E1 -9637.074,E2 -9637.074} C_VEL
LIN {X 0,Y 426.576,Z 103.662,A -85,B 0,C 180,E1 -9638.095,E2 -9638.095} C_VEL
LIN {X 0,Y 425.495,Z 103.792,A -85,B 0,C 180,E1 -9638.885,E2 -9638.885} C_VEL
LIN {X 0,Y 425.404,Z 103.804,A -85,B 0,C 180,E1 -9639.153,E2 -9639.153} C_VEL
LIN {X 0,Y 425.395,Z 103.804,A -85,B 0,C 180,E1 -9642.904,E2 -9642.904} C_VEL
LIN {X 0,Y 425.363,Z 103.808,A -85,B 0,C 180,E1 -9646.606,E2 -9646.606} C_VEL
LIN {X 0,Y 425.331,Z 103.819,A -85,B 0,C 180,E1 -9649.636,E2 -9649.636} C_VEL
LIN {X 0,Y 425.307,Z 103.819,A -85,B 0,C 180,E1 -9653.366,E2 -9653.366} C_VEL
LIN {X 0,Y 425.35,Z 103.81,A -85,B 0,C 180,E1 -9656.845,E2 -9656.845} C_VEL
LIN {X 0,Y 425.293,Z 103.822,A -85,B 0,C 180,E1 -9659.72,E2 -9659.72} C_VEL
LIN {X 0,Y 425.285,Z 103.82,A -85,B 0,C 180,E1 -9663.048,E2 -9663.048} C_VEL
LIN {X 0,Y 425.284,Z 103.82,A -85,B 0,C 180,E1 -9665.929,E2 -9665.929} C_VEL
LIN {X 0,Y 425.3,Z 103.82,A -85,B 0,C 180,E1 -9669.044,E2 -9669.044} C_VEL
LIN {X 0,Y 425.281,Z 103.819,A -85,B 0,C 180,E1 -9672.653,E2 -9672.653} C_VEL
LIN {X 0,Y 425.264,Z 103.821,A -85,B 0,C 180,E1 -9676.044,E2 -9676.044} C_VEL
LIN {X 0,Y 425.277,Z 103.82,A -85,B 0,C 180,E1 -9678.622,E2 -9678.622} C_VEL
LIN {X 0,Y 425.305,Z 103.822,A -85,B 0,C 180,E1 -9681.102,E2 -9681.102} C_VEL
LIN {X 0,Y 425.303,Z 103.821,A -85,B 0,C 180,E1 -9684.664,E2 -9684.664} C_VEL
LIN {X 0,Y 425.289,Z 103.822,A -85,B 0,C 180,E1 -9688.171,E2 -9688.171} C_VEL
LIN {X 0,Y 426.495,Z 106.983,A -85,B 0,C 180,E1 -9688.343,E2 -9688.343} C_VEL
LIN {X 0,Y 441.029,Z 135.894,A -85,B 0,C 180,E1 -9690.001,E2 -9690.001} C_VEL
LIN {X 0,Y 436.84,Z 282.294,A -85,B 0,C 180,E1 -9692.903,E2 -9692.903} C_VEL
LIN {X 0,Y 436.267,Z 301.441,A -85,B 0,C 180,E1 -9693.35,E2 -9693.35} C_VEL
LIN {X 0,Y 435.536,Z 318.675,A -85,B 0,C 180,E1 -9693.946,E2 -9693.946} C_VEL
LIN {X 0,Y 434.618,Z 335.708,A -85,B 0,C 180,E1 -9694.741,E2 -9694.741} C_VEL
LIN {X 0,Y 433.701,Z 350.241,A -85,B 0,C 180,E1 -9695.593,E2 -9695.593} C_VEL
LIN {X 0,Y 432.529,Z 365.367,A -85,B 0,C 180,E1 -9696.668,E2 -9696.668} C_VEL
LIN {X 0,Y 431.285,Z 380.629,A -85,B 0,C 180,E1 -9697.988,E2 -9697.988} C_VEL
LIN {X 0,Y 430.091,Z 393.42,A -85,B 0,C 180,E1 -9699.306,E2 -9699.306} C_VEL
LIN {X 0,Y 428.914,Z 406.322,A -85,B 0,C 180,E1 -9700.87,E2 -9700.87} C_VEL
LIN {X 0,Y 427.852,Z 418.404,A -85,B 0,C 180,E1 -9702.604,E2 -9702.604} C_VEL
LIN {X 0,Y 426.981,Z 428.148,A -85,B 0,C 180,E1 -9704.241,E2 -9704.241} C_VEL
LIN {X 0,Y 426.147,Z 437.819,A -85,B 0,C 180,E1 -9706.165,E2 -9706.165} C_VEL
LIN {X 0,Y 425.531,Z 445.807,A -85,B 0,C 180,E1 -9708.086,E2 -9708.086} C_VEL
LIN {X 0,Y 425.068,Z 452.403,A -85,B 0,C 180,E1 -9710.002,E2 -9710.002} C_VEL
LIN {X 0,Y 424.786,Z 457.777,A -85,B 0,C 180,E1 -9711.916,E2 -9711.916} C_VEL
LIN {X 0,Y 424.671,Z 460.983,A -85,B 0,C 180,E1 -9713.348,E2 -9713.348} C_VEL
LIN {X 0,Y 424.441,Z 464.371,A -85,B 0,C 180,E1 -9715.251,E2 -9715.251} C_VEL
LIN {X 0,Y 424.444,Z 466.622,A -85,B 0,C 180,E1 -9717.153,E2 -9717.153} C_VEL
LIN {X 0,Y 424.275,Z 467.96,A -85,B 0,C 180,E1 -9719.051,E2 -9719.051} C_VEL
LIN {X 0,Y 424.277,Z 468.198,A -85,B 0,C 180,E1 -9720.949,E2 -9720.949} C_VEL
LIN {X 0,Y 424.537,Z 467.474,A -85,B 0,C 180,E1 -9722.847,E2 -9722.847} C_VEL
LIN {X 0,Y 424.607,Z 465.728,A -85,B 0,C 180,E1 -9724.747,E2 -9724.747} C_VEL
LIN {X 0,Y 424.818,Z 462.384,A -85,B 0,C 180,E1 -9726.965,E2 -9726.965} C_VEL
LIN {X 0,Y 425.182,Z 457.951,A -85,B 0,C 180,E1 -9729.034,E2 -9729.034} C_VEL
LIN {X 0,Y 425.679,Z 452.692,A -85,B 0,C 180,E1 -9730.945,E2 -9730.945} C_VEL
LIN {X 0,Y 426.25,Z 446.085,A -85,B 0,C 180,E1 -9732.861,E2 -9732.861} C_VEL
LIN {X 0,Y 427.093,Z 438.077,A -85,B 0,C 180,E1 -9734.777,E2 -9734.777} C_VEL
LIN {X 0,Y 428.121,Z 428.45,A -85,B 0,C 180,E1 -9736.695,E2 -9736.695} C_VEL
LIN {X 0,Y 429.205,Z 418.629,A -85,B 0,C 180,E1 -9738.348,E2 -9738.348} C_VEL
LIN {X 0,Y 430.53,Z 406.694,A -85,B 0,C 180,E1 -9740.048,E2 -9740.048} C_VEL
LIN {X 0,Y 431.854,Z 394.06,A -85,B 0,C 180,E1 -9741.562,E2 -9741.562} C_VEL
LIN {X 0,Y 433.259,Z 380.678,A -85,B 0,C 180,E1 -9742.911,E2 -9742.911} C_VEL
LIN {X 0,Y 434.575,Z 366.721,A -85,B 0,C 180,E1 -9744.101,E2 -9744.101} C_VEL
LIN {X 0,Y 435.833,Z 352.086,A -85,B 0,C 180,E1 -9745.142,E2 -9745.142} C_VEL
LIN {X 0,Y 437.035,Z 336.336,A -85,B 0,C 180,E1 -9746.054,E2 -9746.054} C_VEL
LIN {X 0,Y 437.959,Z 320.366,A -85,B 0,C 180,E1 -9746.796,E2 -9746.796} C_VEL
LIN {X 0,Y 438.791,Z 303.323,A -85,B 0,C 180,E1 -9747.386,E2 -9747.386} C_VEL
LIN {X 0,Y 440.267,Z 269.37,A -85,B 0,C 180,E1 -9748.196,E2 -9748.196} C_VEL
LIN {X 0,Y 444.093,Z 199.849,A -85,B 0,C 180,E1 -9749.901,E2 -9749.901} C_VEL
LIN {X 0,Y 448.253,Z 140.301,A -85,B 0,C 180,E1 -9751.453,E2 -9751.453} C_VEL
LIN {X 0,Y 444.184,Z 132.616,A -85,B 0,C 180,E1 -9752.302,E2 -9752.302} C_VEL
LIN {X 0,Y 439.655,Z 125.006,A -85,B 0,C 180,E1 -9753.321,E2 -9753.321} C_VEL
LIN {X 0,Y 437.678,Z 122.013,A -85,B 0,C 180,E1 -9753.793,E2 -9753.793} C_VEL
LIN {X 0,Y 434.377,Z 117.359,A -85,B 0,C 180,E1 -9754.634,E2 -9754.634} C_VEL
LIN {X 0,Y 431.413,Z 113.595,A -85,B 0,C 180,E1 -9755.458,E2 -9755.458} C_VEL
LIN {X 0,Y 427.644,Z 109.506,A -85,B 0,C 180,E1 -9756.629,E2 -9756.629} C_VEL
LIN {X 0,Y 426.876,Z 107.476,A -85,B 0,C 180,E1 -9757.789,E2 -9757.789} C_VEL
LIN {X 0,Y 425.56,Z 105.085,A -85,B 0,C 180,E1 -9760.096,E2 -9760.096} C_VEL
LIN {X 0,Y 425.353,Z 104.152,A -85,B 0,C 180,E1 -9761.967,E2 -9761.967} C_VEL
LIN {X 0,Y 425.452,Z 104.729,A -85,B 0,C 180,E1 -9763.931,E2 -9763.931} C_VEL
LIN {X 0,Y 426.687,Z 107.287,A -85,B 0,C 180,E1 -9766.446,E2 -9766.446} C_VEL
LIN {X 0,Y 427.71,Z 109.269,A -85,B 0,C 180,E1 -9767.682,E2 -9767.682} C_VEL
LIN {X 0,Y 429.184,Z 112.257,A -85,B 0,C 180,E1 -9769.079,E2 -9769.079} C_VEL
LIN {X 0,Y 431.198,Z 116.773,A -85,B 0,C 180,E1 -9770.731,E2 -9770.731} C_VEL
LIN {X 0,Y 433.778,Z 123.151,A -85,B 0,C 180,E1 -9772.55,E2 -9772.55} C_VEL
LIN {X 0,Y 436.602,Z 130.868,A -85,B 0,C 180,E1 -9774.349,E2 -9774.349} C_VEL
LIN {X 0,Y 438.599,Z 137.087,A -85,B 0,C 180,E1 -9775.556,E2 -9775.556} C_VEL
LIN {X 0,Y 442.414,Z 145.441,A -85,B 0,C 180,E1 -9776.488,E2 -9776.488} C_VEL
LIN {X 0,Y 444.434,Z 161.544,A -85,B 0,C 180,E1 -9777.39,E2 -9777.39} C_VEL
LIN {X 0,Y 446.132,Z 181.924,A -85,B 0,C 180,E1 -9778.321,E2 -9778.321} C_VEL
LIN {X 0,Y 446.343,Z 187.422,A -85,B 0,C 180,E1 -9778.531,E2 -9778.531} C_VEL
LIN {X 0,Y 441.477,Z 267.471,A -85,B 0,C 180,E1 -9780.527,E2 -9780.527} C_VEL
LIN {X 0,Y 437.576,Z 355.484,A -85,B 0,C 180,E1 -9782.596,E2 -9782.596} C_VEL
LIN {X 0,Y 436.224,Z 373.462,A -85,B 0,C 180,E1 -9783.185,E2 -9783.185} C_VEL
LIN {X 0,Y 434.899,Z 390.408,A -85,B 0,C 180,E1 -9783.937,E2 -9783.937} C_VEL
LIN {X 0,Y 433.47,Z 406.162,A -85,B 0,C 180,E1 -9784.811,E2 -9784.811} C_VEL
LIN {X 0,Y 431.825,Z 423.37,A -85,B 0,C 180,E1 -9785.991,E2 -9785.991} C_VEL
LIN {X 0,Y 430.337,Z 439.059,A -85,B 0,C 180,E1 -9787.304,E2 -9787.304} C_VEL
LIN {X 0,Y 429.093,Z 452.387,A -85,B 0,C 180,E1 -9788.627,E2 -9788.627} C_VEL
LIN {X 0,Y 427.868,Z 464.948,A -85,B 0,C 180,E1 -9790.072,E2 -9790.072} C_VEL
LIN {X 0,Y 426.779,Z 477.528,A -85,B 0,C 180,E1 -9791.766,E2 -9791.766} C_VEL
LIN {X 0,Y 425.971,Z 487.798,A -85,B 0,C 180,E1 -9793.383,E2 -9793.383} C_VEL
LIN {X 0,Y 425.332,Z 497.449,A -85,B 0,C 180,E1 -9795.16,E2 -9795.16} C_VEL
LIN {X 0,Y 424.824,Z 506.371,A -85,B 0,C 180,E1 -9797.095,E2 -9797.095} C_VEL
LIN {X 0,Y 424.487,Z 513.808,A -85,B 0,C 180,E1 -9799.023,E2 -9799.023} C_VEL
LIN {X 0,Y 424.31,Z 519.798,A -85,B 0,C 180,E1 -9800.946,E2 -9800.946} C_VEL
LIN {X 0,Y 424.323,Z 524.595,A -85,B 0,C 180,E1 -9802.864,E2 -9802.864} C_VEL
LIN {X 0,Y 424.31,Z 527.402,A -85,B 0,C 180,E1 -9804.296,E2 -9804.296} C_VEL
LIN {X 0,Y 424.281,Z 530.21,A -85,B 0,C 180,E1 -9806.2,E2 -9806.2} C_VEL
LIN {X 0,Y 424.352,Z 531.84,A -85,B 0,C 180,E1 -9808.101,E2 -9808.101} C_VEL
LIN {X 0,Y 424.232,Z 532.445,A -85,B 0,C 180,E1 -9809.999,E2 -9809.999} C_VEL
LIN {X 0,Y 424.348,Z 531.947,A -85,B 0,C 180,E1 -9811.898,E2 -9811.898} C_VEL
LIN {X 0,Y 424.282,Z 530.383,A -85,B 0,C 180,E1 -9813.798,E2 -9813.798} C_VEL
LIN {X 0,Y 424.284,Z 527.73,A -85,B 0,C 180,E1 -9815.703,E2 -9815.703} C_VEL
LIN {X 0,Y 424.301,Z 523.91,A -85,B 0,C 180,E1 -9817.614,E2 -9817.614} C_VEL
LIN {X 0,Y 424.312,Z 518.951,A -85,B 0,C 180,E1 -9819.533,E2 -9819.533} C_VEL
LIN {X 0,Y 424.557,Z 512.648,A -85,B 0,C 180,E1 -9821.457,E2 -9821.457} C_VEL
LIN {X 0,Y 424.955,Z 504.961,A -85,B 0,C 180,E1 -9823.387,E2 -9823.387} C_VEL
LIN {X 0,Y 425.571,Z 495.715,A -85,B 0,C 180,E1 -9825.32,E2 -9825.32} C_VEL
LIN {X 0,Y 426.232,Z 486.303,A -85,B 0,C 180,E1 -9826.994,E2 -9826.994} C_VEL
LIN {X 0,Y 427.154,Z 474.874,A -85,B 0,C 180,E1 -9828.713,E2 -9828.713} C_VEL
LIN {X 0,Y 428.195,Z 463.608,A -85,B 0,C 180,E1 -9830.161,E2 -9830.161} C_VEL
LIN {X 0,Y 429.387,Z 450.508,A -85,B 0,C 180,E1 -9831.608,E2 -9831.608} C_VEL
LIN {X 0,Y 430.601,Z 436.352,A -85,B 0,C 180,E1 -9832.933,E2 -9832.933} C_VEL
LIN {X 0,Y 431.987,Z 421.06,A -85,B 0,C 180,E1 -9834.122,E2 -9834.122} C_VEL
LIN {X 0,Y 433.208,Z 406.073,A -85,B 0,C 180,E1 -9835.076,E2 -9835.076} C_VEL
LIN {X 0,Y 434.447,Z 390.029,A -85,B 0,C 180,E1 -9835.898,E2 -9835.898} C_VEL
LIN {X 0,Y 435.393,Z 373.799,A -85,B 0,C 180,E1 -9836.546,E2 -9836.546} C_VEL
LIN {X 0,Y 436.227,Z 357.879,A -85,B 0,C 180,E1 -9837.008,E2 -9837.008} C_VEL
LIN {X 0,Y 441.16,Z 184.607,A -85,B 0,C 180,E1 -9840.47,E2 -9840.47} C_VEL
LIN {X 0,Y 436.424,Z 150.202,A -85,B 0,C 180,E1 -9841.597,E2 -9841.597} C_VEL
LIN {X 0,Y 437.111,Z 141.492,A -85,B 0,C 180,E1 -9842.485,E2 -9842.485} C_VEL
LIN {X 0,Y 436.549,Z 138.574,A -85,B 0,C 180,E1 -9842.836,E2 -9842.836} C_VEL
LIN {X 0,Y 429.948,Z 117.818,A -85,B 0,C 180,E1 -9845.589,E2 -9845.589} C_VEL
LIN {X 0,Y 425.279,Z 103.824,A -85,B 0,C 180,E1 -9847.561,E2 -9847.561} C_VEL
LIN {X 0,Y 425.278,Z 103.826,A -85,B 0,C 180,E1 -9850.52,E2 -9850.52} C_VEL
LIN {X 0,Y 425.312,Z 103.817,A -85,B 0,C 180,E1 -9853.359,E2 -9853.359} C_VEL
LIN {X 0,Y 425.256,Z 103.826,A -85,B 0,C 180,E1 -9856.648,E2 -9856.648} C_VEL
LIN {X 0,Y 425.29,Z 103.82,A -85,B 0,C 180,E1 -9859.873,E2 -9859.873} C_VEL
LIN {X 0,Y 425.28,Z 103.824,A -85,B 0,C 180,E1 -9862.487,E2 -9862.487} C_VEL
LIN {X 0,Y 425.303,Z 103.818,A -85,B 0,C 180,E1 -9865.817,E2 -9865.817} C_VEL
LIN {X 0,Y 425.296,Z 103.817,A -85,B 0,C 180,E1 -9869.236,E2 -9869.236} C_VEL
LIN {X 0,Y 425.345,Z 103.814,A -85,B 0,C 180,E1 -9872.442,E2 -9872.442} C_VEL
LIN {X 0,Y 425.347,Z 103.813,A -85,B 0,C 180,E1 -9875.602,E2 -9875.602} C_VEL
LIN {X 0,Y 425.288,Z 103.818,A -85,B 0,C 180,E1 -9878.681,E2 -9878.681} C_VEL
LIN {X 0,Y 425.329,Z 103.817,A -85,B 0,C 180,E1 -9881.703,E2 -9881.703} C_VEL
LIN {X 0,Y 425.351,Z 103.81,A -85,B 0,C 180,E1 -9884.671,E2 -9884.671} C_VEL
LIN {X 0,Y 425.425,Z 103.805,A -85,B 0,C 180,E1 -9887.599,E2 -9887.599} C_VEL
LIN {X 0,Y 425.438,Z 103.802,A -85,B 0,C 180,E1 -9891.45,E2 -9891.45} C_VEL
LIN {X 0,Y 425.55,Z 103.786,A -85,B 0,C 180,E1 -9894.313,E2 -9894.313} C_VEL
LIN {X 0,Y 425.571,Z 103.785,A -85,B 0,C 180,E1 -9898.107,E2 -9898.107} C_VEL
LIN {X 0,Y 425.699,Z 103.769,A -85,B 0,C 180,E1 -9900,E2 -9900} C_VEL
LIN {X 0,Y 425.553,Z 103.785,A -85,B 0,C 180,E1 -9902.84,E2 -9902.84} C_VEL
LIN {X 0,Y 425.526,Z 103.788,A -85,B 0,C 180,E1 -9906.639,E2 -9906.639} C_VEL
